# B&R Automation Studio project Panasonic_LinkaPowerCP2_A2021055 (part 15)

#### Main.st - Init, cyclic, exit code
```iecst
PROGRAM _INIT
	(* Insert code here *)

END_PROGRAM

PROGRAM _CYCLIC

	//*************************************Prepnutie obrazovky pri stlačení tlačítka CS*********************************//
	IF EDGEPOS(P1_Pracovisko.STAV.Manual AND NOT Safety.STAV.Linka_ZonaCS_AKTIVNA) THEN
		P1_Vizu.GoPage:= 'PageAutomatP1';
	END_IF

	//************************************Filter alarmov**************************************************************//
	FilterVizu_P1:= '[{"logicalOperator":"and","value":100,"conditionType":">=","columnType":"cod","useAlarmState":false,"alarmState":0},{"value":199,"conditionType":"<=","columnType":"cod","useAlarmState":false,"alarmState":0}]';

	//Zmeny farieb tlačítok ovládania zámkov//
	//Predné dvere //
	IF P1_Pracovisko.OUT.PredneDvere_ZAMKNI AND P1_Pracovisko.IN.PredneDvere_PritomnostAdaptera THEN
		P1_Vizu.TL_PrednyZamok_Farba:= "Button_Green";
	ELSIF P1_Pracovisko.IN.PredneDvere_PritomnostAdaptera THEN
		IF Blikac1s THEN
			P1_Vizu.TL_PrednyZamok_Farba:= "Button_Blue";
		ELSE
			P1_Vizu.TL_PrednyZamok_Farba:= "Operate";
		END_IF
	ELSE
		P1_Vizu.TL_PrednyZamok_Farba:= "Button_Red";
	END_IF

	//Zadné dvere//
	IF P1_Pracovisko.OUT.ZadneDvere_ZAMKNI AND P1_Pracovisko.IN.ZadneDvere_PritomnostAdaptera THEN
		P1_Vizu.TL_ZadnyZamok_Farba:= "Button_Green";
	ELSIF P1_Pracovisko.IN.ZadneDvere_PritomnostAdaptera THEN
		IF Blikac1s THEN
			P1_Vizu.TL_ZadnyZamok_Farba:= "Button_Blue";
		ELSE
			P1_Vizu.TL_ZadnyZamok_Farba:= "Operate";
		END_IF
	ELSE
		P1_Vizu.TL_ZadnyZamok_Farba:= "Button_Red";
	END_IF

	//***********************************Zobrazenie warningov pracoviska****************************************************//
	//0 - Pracovisko je vypnuté.
	//1 - Prebieha inicializácia pracoviska.
	//2 - Na pracovisku prebieha výroba.
	//3 - Prebieha ukončenie pracovného cyklu pracoviska.
	//4 - Prebieha režim vyprázdnenia linky.
	//5 - Robot nie je prepnuty do automatického režimu !!!
	//6 - Doplň zásobník skrutiek K30 !!!
	//7 - Doplň zásobník skrutiek M5 !!!
	//8 - Doplň zásobník skrutiek M4 !!!
	//10 - Testovací kus

	IF NOT P1_Robot.COM_IN.Stav_RezimAUTOMAT THEN
		P1_Vizu.Warnings_Index:= 5;
	ELSIF P1_Pracovisko.STAV.Automat AND NOT P1_Pracovisko.STAV.PoINIT AND NOT P1_Pracovisko.STAV.UkoncenieCyklu_BUSY THEN
		P1_Vizu.Warnings_Index:= 1;
	ELSIF P1_Srobovanie.SkrutSet_K30.IN.VibracnyHrniec.PritomnostSkrutiekVHrnci THEN
		P1_Vizu.Warnings_Index:= 6;
	ELSIF P1_Srobovanie.SkrutSet_M5.IN.ZasobnikSkrutiekPrazdny THEN
		P1_Vizu.Warnings_Index:= 7;
	ELSIF P1_Srobovanie.SkrutSet_M4.IN.ZasobnikSkrutiekPrazdny THEN
		P1_Vizu.Warnings_Index:= 8;
	ELSIF Linka.PAR.TestovaciKus THEN
		P1_Vizu.Warnings_Index:= 10;
	ELSIF Linka.PAR.VyprazdnenieLinky THEN
		P1_Vizu.Warnings_Index:= 4;
	ELSIF P1_Pracovisko.STAV.PoINIT AND NOT P1_Pracovisko.STAV.UkoncenieCyklu_BUSY THEN
		P1_Vizu.Warnings_Index:= 2;
	ELSIF P1_Pracovisko.STAV.UkoncenieCyklu_BUSY THEN
		P1_Vizu.Warnings_Index:= 3;
	ELSIF NOT P1_Pracovisko.STAV.Automat THEN
		P1_Vizu.Warnings_Index:= 0;
	END_IF

	//************************Prepínanie farby textového pola warning zariadenia***********************************//
	IF P1_Vizu.Warnings_Index = 0 THEN
		P1_Vizu.Warnings_Farba:= "TextOutput_Grey";
	ELSIF P1_Vizu.Warnings_Index = 1 THEN
		P1_Vizu.Warnings_Farba:= "TextOutput_Blue";
	ELSIF P1_Vizu.Warnings_Index = 2 THEN
		P1_Vizu.Warnings_Farba:= "TextOutput_Green";
	ELSIF P1_Vizu.Warnings_Index = 3 THEN
		P1_Vizu.Warnings_Farba:= "TextOutput_Blue";
	ELSIF P1_Vizu.Warnings_Index = 4 THEN
		P1_Vizu.Warnings_Farba:= "TextOutput_Green";
	ELSIF P1_Vizu.Warnings_Index = 10 THEN
		P1_Vizu.Warnings_Farba:= "TextOutput_Green";
	ELSE
		IF Blikac1s THEN
			P1_Vizu.Warnings_Farba:= "TextOutput_Orange";
		ELSE
			P1_Vizu.Warnings_Farba:= "TextOutput_Grey";
		END_IF
	END_IF

	//***********************Prepnutie bootovacej obrazovky********************************//
	IF P1_Vizu.ActualPage <> 'PageBootP1' AND NOT Safety.STAV.Linka_SafetyPLC_Nabehlo THEN
		P1_Vizu.GoPage:= 'PageBootP1';
	ELSIF P1_Vizu.ActualPage = 'PageBootP1' AND Safety.STAV.Linka_SafetyPLC_Nabehlo THEN
		P1_Vizu.GoPage:= 'PageAutomatP1';
	END_IF

	IF P1_Vizu.GoPage = 'PageBootP1' AND P1_Vizu.ActualPage = 'PageBootP1' THEN
		P1_Vizu.GoPage:= '';
	ELSIF P1_Vizu.GoPage = 'PageAutomatP1' AND P1_Vizu.ActualPage = 'PageAutomatP1' THEN
		P1_Vizu.GoPage:= '';
	END_IF

	//********************************Blikanie tlačítka Alarmy*******************************************************//
	IF P1_Pracovisko.STAV.PORUCHA AND P1_Vizu.ActualPage <> 'PageAlarmP1' THEN
		IF Blikac500ms THEN
			P1_AlarmyVizu.FarbaTlacitka_Alarmy:= "Button_Red";
		ELSE
			P1_AlarmyVizu.FarbaTlacitka_Alarmy:= "default";
		END_IF
	ELSE
		P1_AlarmyVizu.FarbaTlacitka_Alarmy:= "default";
	END_IF

	//*************************************Zamknutie tlačítok***************************************************************//
	//Zamknutie tlačítok ovládania zámkov//
	IF P1_Pracovisko.STAV.Automat THEN
		P1_Vizu.TL_OvladaniaZamkov_ENABLE:= FALSE;
	ELSIF P1_Srobovanie.STAV.RR_Polohovanie_BUSY THEN
		P1_Vizu.TL_OvladaniaZamkov_ENABLE:= FALSE;
	ELSIF P1_Srobovanie.STAV.CistenieSkrutkovackyK30_BUSY THEN
		P1_Vizu.TL_OvladaniaZamkov_ENABLE:= FALSE;
	ELSE
		P1_Vizu.TL_OvladaniaZamkov_ENABLE:= TRUE;
	END_IF

	//Tlačítko Štat Automat//
	IF P1_Pracovisko.STAV.UkoncenieCyklu_BUSY THEN
		P1_Vizu.TL_StartAutomat_ENABLE:= FALSE;
	ELSIF P1_Pracovisko.STAV.PORUCHA THEN
		P1_Vizu.TL_StartAutomat_ENABLE:= FALSE;
	ELSIF NOT P1_Robot.COM_IN.Stav_RezimAUTOMAT THEN
		P1_Vizu.TL_StartAutomat_ENABLE:= FALSE;
	ELSIF NOT Safety.STAV.P1_ZonaBunky_AKTIVNA THEN
		P1_Vizu.TL_StartAutomat_ENABLE:= FALSE;
	ELSIF NOT P1_Pracovisko.STAV.HardwareVytahu_OK THEN
		P1_Vizu.TL_StartAutomat_ENABLE:= FALSE;
	ELSIF NOT P1_Pracovisko.STAV.HardwareBunky_OK THEN
		P1_Vizu.TL_StartAutomat_ENABLE:= FALSE;
	ELSE
		P1_Vizu.TL_StartAutomat_ENABLE:= TRUE;
	END_IF

	//Tlačítko Ukončenie Cyklu//
	IF P1_Pracovisko.STAV.PoINIT THEN
		P1_Vizu.TL_KoniecCyklu_ENABLE:= TRUE;
	ELSE
		P1_Vizu.TL_KoniecCyklu_ENABLE:= FALSE;
	END_IF

	//Tlačítko STOP//
	IF P1_Pracovisko.STAV.PoINIT AND NOT P1_Pracovisko.STAV.UkoncenieCyklu_BUSY THEN
		P1_Vizu.TL_STOP_ENABLE:= FALSE;
	ELSE
		P1_Vizu.TL_STOP_ENABLE:= TRUE;
	END_IF

	//Tlačítko Režim Automat//

	P1_Vizu.TL_RezimAutomat_ENABLE:= TRUE;

	//Tlačítko Režim Manual//
	IF P1_Pracovisko.STAV.Automat THEN
		P1_Vizu.TL_RezimManual_ENABLE:= FALSE;
	ELSIF NOT P1_Pracovisko.STAV.HardwareVytahu_OK THEN
		P1_Vizu.TL_RezimManual_ENABLE:= FALSE;
	ELSIF NOT P1_Pracovisko.STAV.HardwareBunky_OK THEN
		P1_Vizu.TL_RezimManual_ENABLE:= FALSE;
	ELSE
		P1_Vizu.TL_RezimManual_ENABLE:= TRUE;
	END_IF

	//Tlačítko zmena modelu//
	IF Linka.STAV.OFF THEN
		P1_Vizu.TL_VolbaModelu_ENABLE:= TRUE;
	ELSE
		P1_Vizu.TL_VolbaModelu_ENABLE:= FALSE;
	END_IF

	//Tlačítko paletka prechádza//
	IF NOT Linka.STAV.PoINIT THEN
		P1_Vizu.TL_PaletkaPrechadza_ENABLE:= FALSE;
	ELSIF NOT P1_Vytah.RFID_hlava.PritomnostPaletky THEN
		P1_Vizu.TL_PaletkaPrechadza_ENABLE:= FALSE;
	ELSIF Linka.PAR.TestovaciKus THEN
		P1_Vizu.TL_PaletkaPrechadza_ENABLE:= FALSE;
	ELSIF Linka.PAR.RevorkovyKus THEN
		P1_Vizu.TL_PaletkaPrechadza_ENABLE:= FALSE;
	ELSIF Linka.PAR.PaletkaPrechadza THEN
		P1_Vizu.TL_PaletkaPrechadza_ENABLE:= FALSE;
	ELSE
		P1_Vizu.TL_PaletkaPrechadza_ENABLE:= TRUE;
	END_IF

	//Tlačítko vyprázdnenie linky//
	IF Linka.PAR.VyprazdnenieLinky THEN
		P1_Vizu.TL_VyprazdnenieLinky_ENABLE:= FALSE;
	ELSIF NOT P4_Pracovisko.STAV.Automat THEN
		P1_Vizu.TL_VyprazdnenieLinky_ENABLE:= FALSE;
	ELSIF Linka.PAR.TestovaciKus THEN
		P1_Vizu.TL_VyprazdnenieLinky_ENABLE:= FALSE;
	ELSE
		P1_Vizu.TL_VyprazdnenieLinky_ENABLE:= TRUE;
	END_IF

	//Tlačítko testovací kus//
	IF NOT Linka.STAV.PoINIT THEN
		P1_Vizu.TL_TestovaciKus_ENABLE:= FALSE;
	ELSIF Linka.PAR.RevorkovyKus THEN
		P1_Vizu.TL_TestovaciKus_ENABLE:= FALSE;
	ELSIF NOT P1_Vytah.RFID_hlava.PritomnostPaletky THEN
		P1_Vizu.TL_TestovaciKus_ENABLE:= FALSE;
	ELSIF Linka.PAR.PaletkaPrechadza THEN
		P1_Vizu.TL_TestovaciKus_ENABLE:= FALSE;
	ELSE
		P1_Vizu.TL_TestovaciKus_ENABLE:= TRUE;
	END_IF

	//Tlačítko revork//
	IF NOT Linka.STAV.PoINIT THEN
		P1_Vizu.TL_Revork_ENABLE:= FALSE;
	ELSIF NOT P1_Vytah.RFID_hlava.PritomnostPaletky THEN
		P1_Vizu.TL_Revork_ENABLE:= FALSE;
	ELSIF Linka.PAR.TestovaciKus THEN
		P1_Vizu.TL_Revork_ENABLE:= FALSE;
	ELSIF Linka.PAR.PaletkaPrechadza THEN
		P1_Vizu.TL_Revork_ENABLE:= FALSE;
	ELSE
		P1_Vizu.TL_Revork_ENABLE:= TRUE;
	END_IF

	//Tlačítko výtah čítanie paletky//
	IF P1_Vytah.RFID_hlava.PritomnostPaletky THEN
		P1_Vizu.Vytah_CitaniePaletky_ENABLE:= TRUE;
	ELSE
		P1_Vizu.Vytah_CitaniePaletky_ENABLE:= FALSE;
	END_IF

	//Tlačítko výťah zápis paletky//
	IF P1_Vytah.RFID_hlava.PritomnostPaletky THEN
		P1_Vizu.Vytah_ZapisPaletky_ENABLE:= TRUE;
	ELSE
		P1_Vizu.Vytah_ZapisPaletky_ENABLE:= FALSE;
	END_IF

	//RR - Tlačítko čistenia skrutkovačky K30//
	IF P1_Srobovanie.STAV.RR_Polohovanie_BUSY THEN
		P1_Vizu.TL_VycistiSkrutkovackuK30_ENABLE:= FALSE;
	ELSIF NOT Safety.STAV.P1_ZonaBunky_AKTIVNA THEN
		P1_Vizu.TL_VycistiSkrutkovackuK30_ENABLE:= FALSE;
	ELSIF NOT Safety.STAV.Linka_ZonaCS_AKTIVNA THEN
		P1_Vizu.TL_VycistiSkrutkovackuK30_ENABLE:= FALSE;
	ELSIF P1_Srobovanie.STAV.CistenieSkrutkovackyK30_BUSY THEN
		P1_Vizu.TL_VycistiSkrutkovackuK30_ENABLE:= FALSE;
	ELSIF NOT P1_Pracovisko.STAV.SkrutkovackyZasunute THEN
		P1_Vizu.TL_VycistiSkrutkovackuK30_ENABLE:= FALSE;
	ELSIF P1_Srobovanie.CMD.RR_SkrutSetK30_VysunBrzdu THEN
		P1_Vizu.TL_VycistiSkrutkovackuK30_ENABLE:= FALSE;
	ELSIF P1_Srobovanie.CMD.RR_SkrutSetK30_Zasobnik_RUN THEN
		P1_Vizu.TL_VycistiSkrutkovackuK30_ENABLE:= FALSE;
	ELSE
		P1_Vizu.TL_VycistiSkrutkovackuK30_ENABLE:= TRUE;
	END_IF

	//RR - Tlačítko polohovania aplikátora//
	IF P1_Srobovanie.STAV.RR_Polohovanie_BUSY THEN
		P1_Vizu.TL_PolohujManipulator_ENABLE:= FALSE;
	ELSIF NOT Safety.STAV.P1_ZonaBunky_AKTIVNA THEN
		P1_Vizu.TL_PolohujManipulator_ENABLE:= FALSE;
	ELSIF NOT Safety.STAV.Linka_ZonaCS_AKTIVNA THEN
		P1_Vizu.TL_PolohujManipulator_ENABLE:= FALSE;
	ELSIF P1_Srobovanie.STAV.CistenieSkrutkovackyK30_BUSY THEN
		P1_Vizu.TL_PolohujManipulator_ENABLE:= FALSE;
	ELSIF NOT P1_Pracovisko.STAV.SkrutkovackyZasunute THEN
		P1_Vizu.TL_PolohujManipulator_ENABLE:= FALSE;
	ELSE
		P1_Vizu.TL_PolohujManipulator_ENABLE:= TRUE;
	END_IF

	//RR - Tlačítko vysunutia skrutkovačky K30//
	IF P1_Srobovanie.STAV.RR_Polohovanie_BUSY THEN
		P1_Vizu.Tl_VysunutieSkrutkovK30_ENABLE:= FALSE;
	ELSIF P1_Srobovanie.STAV.CistenieSkrutkovackyK30_BUSY THEN
		P1_Vizu.Tl_VysunutieSkrutkovK30_ENABLE:= FALSE;
	ELSIF NOT Safety.STAV.P1_ZonaBunky_AKTIVNA THEN
		P1_Vizu.Tl_VysunutieSkrutkovK30_ENABLE:= FALSE;
	ELSIF NOT Safety.STAV.Linka_ZonaCS_AKTIVNA THEN
		P1_Vizu.Tl_VysunutieSkrutkovK30_ENABLE:= FALSE;
	ELSE
		P1_Vizu.Tl_VysunutieSkrutkovK30_ENABLE:= TRUE;
	END_IF

	//RR - Tlačítko vysunutia skrutkovačiek M4 a M5//
	IF P1_Srobovanie.STAV.RR_Polohovanie_BUSY THEN
		P1_Vizu.TL_OvladaniaVysunSkrutkovM4_M5:= FALSE;
	ELSIF P1_Srobovanie.STAV.CistenieSkrutkovackyK30_BUSY THEN
		P1_Vizu.TL_OvladaniaVysunSkrutkovM4_M5:= FALSE;
	ELSIF NOT Safety.STAV.P1_ZonaBunky_AKTIVNA THEN
		P1_Vizu.TL_OvladaniaVysunSkrutkovM4_M5:= FALSE;
	ELSIF NOT Safety.STAV.Linka_ZonaCS_AKTIVNA THEN
		P1_Vizu.TL_OvladaniaVysunSkrutkovM4_M5:= FALSE;
	ELSE
		P1_Vizu.TL_OvladaniaVysunSkrutkovM4_M5:= TRUE;
	END_IF

	//RR - Ovládanie skrutkovacieho setu//
	IF P1_Srobovanie.STAV.CistenieSkrutkovackyK30_BUSY THEN
		P1_Vizu.TL_OvladSkrutkovSetuK30_ENABLE:= FALSE;
	ELSE
		P1_Vizu.TL_OvladSkrutkovSetuK30_ENABLE:= TRUE;
	END_IF

	//RR - Ovládanie manipulatora XY//
	IF NOT Safety.STAV.P1_ZonaBunky_AKTIVNA THEN
		P1_Vizu.TL_OvladManipulatoraXY_ENABLE:= FALSE;
	ELSE
		P1_Vizu.TL_OvladManipulatoraXY_ENABLE:= TRUE;
	END_IF

	//**************************Zamknutie editácie parametrov*********************************//
	IF P1_UrovenPrihlasenehoUzivatela >= 20 THEN
		P1_Vizu.EditaciaParametrov_ENABLE:= TRUE;
	ELSE
		P1_Vizu.EditaciaParametrov_ENABLE:= FALSE;
	END_IF

	//***********************************Prepínanie stavov pracovísk*******************************************************************//
	//Výťah//
	IF NOT P1_Pracovisko.STAV.HardwareVytahu_OK THEN
		P1_Vizu.IndexStavu_Vytah:= 3;
	ELSIF P1_Pracovisko.STAV.Porucha_ST1 THEN
		P1_Vizu.IndexStavu_Vytah:= 3;
	ELSIF P1_Vytah.Automat AND NOT P1_Vytah.STAV.PoINIT THEN
		P1_Vizu.IndexStavu_Vytah:= 1;
	ELSIF P1_Vytah.Automat AND P1_Vytah.STAV.PoINIT THEN
		P1_Vizu.IndexStavu_Vytah:= 2;
	ELSE
		P1_Vizu.IndexStavu_Vytah:= 0;
	END_IF

	//Dopravníky//
	IF P1_Dopravniky.Automat AND NOT P1_Dopravniky.STAV.PoINIT THEN
		P1_Vizu.IndexStavu_Dopravnik:= 1;
	ELSIF P1_Dopravniky.Automat AND P1_Dopravniky.STAV.PoINIT THEN
		P1_Vizu.IndexStavu_Dopravnik:= 2;
	ELSE
		P1_Vizu.IndexStavu_Dopravnik:= 0;
	END_IF

	//Spodný stoper//
	IF P1_SpodnyStoper.Automat AND NOT P1_SpodnyStoper.STAV.PoINIT THEN
		P1_Vizu.IndexStavu_SpodnyStoper:= 1;
	ELSIF P1_SpodnyStoper.Automat AND P1_SpodnyStoper.STAV.PoINIT THEN
		P1_Vizu.IndexStavu_SpodnyStoper:= 2;
	ELSE
		P1_Vizu.IndexStavu_SpodnyStoper:= 0;
	END_IF

	//Stoper šrobovania//
	IF NOT P1_Pracovisko.STAV.HardwareBunky_OK THEN
		P1_Vizu.IndexStavu_StoperSrobovania:= 3;
	ELSIF P1_Pracovisko.STAV.Porucha_ST2 THEN
		P1_Vizu.IndexStavu_StoperSrobovania:= 3;
	ELSIF P1_StoperSrobovania.Automat AND NOT P1_StoperSrobovania.STAV.PoINIT THEN
		P1_Vizu.IndexStavu_StoperSrobovania:= 1;
	ELSIF P1_StoperSrobovania.Automat AND P1_StoperSrobovania.STAV.PoINIT THEN
		P1_Vizu.IndexStavu_StoperSrobovania:= 2;
	ELSE
		P1_Vizu.IndexStavu_StoperSrobovania:= 0;
	END_IF

	//Šrobovanie//
	IF NOT P1_Pracovisko.STAV.HardwareBunky_OK THEN
		P1_Vizu.IndexStavu_Srobovanie:= 3;
	ELSIF P1_Pracovisko.STAV.Porucha_ST2 THEN
		P1_Vizu.IndexStavu_Srobovanie:= 3;
	ELSIF P1_Srobovanie.Automat AND NOT P1_Srobovanie.STAV.PoINIT THEN
		P1_Vizu.IndexStavu_Srobovanie:= 1;
	ELSIF P1_Srobovanie.Automat AND P1_Srobovanie.STAV.PoINIT THEN
		P1_Vizu.IndexStavu_Srobovanie:= 2;
	ELSE
		P1_Vizu.IndexStavu_Srobovanie:= 0;
	END_IF

	//Akumulačný stoper//
	IF P1_Pracovisko.STAV.Porucha_ST3 THEN
		P1_Vizu.IndexStavu_AkumulacnyStoper:= 3;
	ELSIF P1_AkumulacnyStoper.Automat AND NOT P1_AkumulacnyStoper.STAV.PoINIT THEN
		P1_Vizu.IndexStavu_AkumulacnyStoper:= 1;
	ELSIF P1_AkumulacnyStoper.Automat AND P1_AkumulacnyStoper.STAV.PoINIT THEN
		P1_Vizu.IndexStavu_AkumulacnyStoper:= 2;
	ELSE
		P1_Vizu.IndexStavu_AkumulacnyStoper:= 0;
	END_IF

	//Robot//
	IF P1_Robot.Automat AND NOT P1_Robot.STAV.PoINIT THEN
		P1_Vizu.IndexStavu_Robot:= 1;
	ELSIF P1_Robot.Automat AND P1_Robot.STAV.PoINIT THEN
		P1_Vizu.IndexStavu_Robot:= 2;
	ELSE
		P1_Vizu.IndexStavu_Robot:= 0;
	END_IF

END_PROGRAM

PROGRAM _EXIT
	(* Insert code here *)

END_PROGRAM
```

### Program Logical/Program/Pracovisko_1/P1_OvladSafety (IEC)

#### Main.st - Init, cyclic, exit code
```iecst
PROGRAM _INIT
	(* Insert code here *)

END_PROGRAM

PROGRAM _CYCLIC

	//******************************************Ovládanie zámkov dverí bunky****************************************//
	//Predné dvere //
	IF P1_Vizu.TL_ZamkniPrednyZamok THEN
		IF NOT P1_Pracovisko.OUT.PredneDvere_ZAMKNI AND P1_Pracovisko.IN.PredneDvere_PritomnostAdaptera THEN
			P1_Pracovisko.OUT.PredneDvere_ZAMKNI:= TRUE;
		ELSIF P1_Pracovisko.OUT.PredneDvere_ZAMKNI THEN
			P1_Pracovisko.OUT.PredneDvere_ZAMKNI:= FALSE;
		END_IF
		P1_Vizu.TL_ZamkniPrednyZamok:= FALSE;
	END_IF

	//Zadné dvere//
	IF P1_Vizu.TL_ZamkniZadnyZamok THEN
		IF NOT P1_Pracovisko.OUT.ZadneDvere_ZAMKNI AND P1_Pracovisko.IN.ZadneDvere_PritomnostAdaptera THEN
			P1_Pracovisko.OUT.ZadneDvere_ZAMKNI:= TRUE;
		ELSIF P1_Pracovisko.OUT.ZadneDvere_ZAMKNI THEN
			P1_Pracovisko.OUT.ZadneDvere_ZAMKNI:= FALSE;
		END_IF
		P1_Vizu.TL_ZamkniZadnyZamok:= FALSE;
	END_IF

	//******************************************Reset zóny výtahu*********************************************//
	IF Safety.STAV.Linka_ZonaCS_AKTIVNA AND
		(Safety.STAV.P1_Vytah_Bariera_AKTIVNA OR Safety.STAV.P1_Vytah_Muting_AKTIVNY) AND
		NOT Safety.STAV.P1_ZonaVytahu_AKTIVNA THEN
		Safety.OUT.P1_ResetZonyVytahu:= TRUE;
	ELSE
		Safety.OUT.P1_ResetZonyVytahu:= FALSE;
	END_IF

	//*****************************************Reset zóny bunky************************************************//
	IF Safety.STAV.Linka_ZonaCS_AKTIVNA AND
		(Safety.STAV.P1_Bunka_Zamky_AKTIVNE OR Safety.STAV.P1_VyblokovanieZamkov_AKTIVNE) AND
		NOT Safety.STAV.P1_ZonaBunky_AKTIVNA AND
		(Safety.STAV.P1_VstupBunky_VstupBar_AKTIVNA OR Safety.STAV.P1_VstupBunky_VystupBar_AKTIVNA) AND
		(Safety.STAV.P1_VystupBunky_VstupBar_AKTIVNA OR Safety.STAV.P1_VystupBunky_VystupBar_AKTIVNA) THEN
		Safety.OUT.P1_ResetZonyBunky:= TRUE;
	ELSE
		Safety.OUT.P1_ResetZonyBunky:= FALSE;
	END_IF

END_PROGRAM

PROGRAM _EXIT
	(* Insert code here *)

END_PROGRAM
```

### Program Logical/Program/Pracovisko_1/P1_Mapping_IO (IEC)

#### Main.st - Init, cyclic, exit code
```iecst
PROGRAM _INIT
	(* Insert code here *)

END_PROGRAM

PROGRAM _CYCLIC

	//**********************************************************IO modul Wedmuller**********************************************************************//
	//************Karta AB 1.2 8DI**************//
	P1_Srobovanie.IN.NapajanieSkrutkovackyK30_OK :=  P1_Pracovisko.COM_Weidmuller.AB1_2_8DI.0;
	P1_Srobovanie.IN.NapajanieSkrutkovackyM5_OK := P1_Pracovisko.COM_Weidmuller.AB1_2_8DI.1;
	P1_Srobovanie.IN.NapajanieSkrutkovackyM4_OK := P1_Pracovisko.COM_Weidmuller.AB1_2_8DI.2;
	P1_Srobovanie.IN.NapajanieZasobnikaM4_OK := P1_Pracovisko.COM_Weidmuller.AB1_2_8DI.3;
	P1_Srobovanie.IN.NapajanieVibrolistyM4_OK := P1_Pracovisko.COM_Weidmuller.AB1_2_8DI.4;
	P1_Srobovanie.IN.NapajanieZasobnikaM5_OK := P1_Pracovisko.COM_Weidmuller.AB1_2_8DI.5;
	P1_Srobovanie.IN.NapajanieVibrolistyM5_OK := P1_Pracovisko.COM_Weidmuller.AB1_2_8DI.6;
	P1_Vytah.IN.StavRiadeniaDopravVytahu_READY := P1_Pracovisko.COM_Weidmuller.AB1_2_8DI.7;

	//***********Karta AB 1.3 8DI***************//
	P1_Dopravniky.IN.StavRiadeniaDopravBunky_READY := P1_Pracovisko.COM_Weidmuller.AB1_3_8DI.0;
	P1_Dopravniky.IN.StavRiadeniaVratnehoDoprav_READY := P1_Pracovisko.COM_Weidmuller.AB1_3_8DI.1;
	P1_Vytah.IN.TeplotaMotoraDopravVytahu_OK := P1_Pracovisko.COM_Weidmuller.AB1_3_8DI.2;
	P1_Dopravniky.IN.TeplotaMotoraDopravBunky_OK := P1_Pracovisko.COM_Weidmuller.AB1_3_8DI.3;
	P1_Dopravniky.IN.TeplotaMotoraVratnehoDoprav_OK := P1_Pracovisko.COM_Weidmuller.AB1_3_8DI.4;
	P1_Pracovisko.COM_Weidmuller.AB1_3_8DI.5;
	P1_Pracovisko.COM_Weidmuller.AB1_3_8DI.6;
	P1_Srobovanie.IN.NapajanieZasobnikaK30_OK := P1_Pracovisko.COM_Weidmuller.AB1_3_8DI.7;

	//************Karta AB 1.4 8DI**************//
	P1_Pracovisko.COM_Weidmuller.AB1_4_8DI.0;
	P1_Pracovisko.COM_Weidmuller.AB1_4_8DI.1;
	P1_Pracovisko.COM_Weidmuller.AB1_4_8DI.2;
	P1_Pracovisko.COM_Weidmuller.AB1_4_8DI.3;
	P1_Pracovisko.COM_Weidmuller.AB1_4_8DI.4;
	P1_Pracovisko.COM_Weidmuller.AB1_4_8DI.5;
	P1_Pracovisko.COM_Weidmuller.AB1_4_8DI.6;
	P1_Pracovisko.COM_Weidmuller.AB1_4_8DI.7;

	//************Karta AB 1.5 8DI***************//
	Safety.IN.Linka_SV_ZonaCS := P1_Pracovisko.COM_Weidmuller.AB1_5_8DI.0;
	Safety.IN.P1_SV_ZonaBunky := P1_Pracovisko.COM_Weidmuller.AB1_5_8DI.1;
	Safety.IN.P1_SV_ZonaVytahu := P1_Pracovisko.COM_Weidmuller.AB1_5_8DI.2;
	P1_Pracovisko.COM_Weidmuller.AB1_5_8DI.3;
	P1_Pracovisko.COM_Weidmuller.AB1_5_8DI.4;
	P1_Pracovisko.COM_Weidmuller.AB1_5_8DI.5;
	P1_Pracovisko.COM_Weidmuller.AB1_5_8DI.6;
	P1_Pracovisko.COM_Weidmuller.AB1_5_8DI.7;

	//************Karta AB 1.6 8DO***************//
	P1_Pracovisko.COM_Weidmuller.AB1_6_8DO.0 := P1_Pracovisko.OUT.Majak_ZeleneSvetlo_ON;
	P1_Pracovisko.COM_Weidmuller.AB1_6_8DO.1 := P1_Pracovisko.OUT.Majak_OranzoveSvetlo_ON;
	P1_Pracovisko.COM_Weidmuller.AB1_6_8DO.2 := P1_Pracovisko.OUT.Majak_CerveneSvetlo_ON;
	P1_Pracovisko.COM_Weidmuller.AB1_6_8DO.3 := P1_Pracovisko.OUT.Majak_Hukacka_ON;
	P1_Pracovisko.COM_Weidmuller.AB1_6_8DO.4 := P1_Srobovanie.SkrutSet_M4.OUT.VibropohonZasobnika_RUN;
	P1_Pracovisko.COM_Weidmuller.AB1_6_8DO.5 := P1_Srobovanie.SkrutSet_M4.OUT.VibropohonListy_RUN;
	P1_Pracovisko.COM_Weidmuller.AB1_6_8DO.6 := P1_Srobovanie.SkrutSet_M5.OUT.VibropohonZasobnika_RUN;
	P1_Pracovisko.COM_Weidmuller.AB1_6_8DO.7 := P1_Srobovanie.SkrutSet_M5.OUT.VibropohonListy_RUN;

	//************Karta AB 1.7 8DO***************//
	P1_Pracovisko.COM_Weidmuller.AB1_7_8DO.0 := P1_Pracovisko.OUT.OsvetlenieBunky_ON;
	P1_Pracovisko.COM_Weidmuller.AB1_7_8DO.1 := P1_Vytah.OUT.DopravnikChod_VPRED;
	P1_Pracovisko.COM_Weidmuller.AB1_7_8DO.2 := P1_Vytah.OUT.DopravnikChod_VZAD;
	P1_Pracovisko.COM_Weidmuller.AB1_7_8DO.3 := P1_Dopravniky.OUT.DopravnikBunky_ON;
	P1_Pracovisko.COM_Weidmuller.AB1_7_8DO.4 := P1_Dopravniky.OUT.VratnyDopravnik_ON;
	P1_Pracovisko.COM_Weidmuller.AB1_7_8DO.5 := P1_Robot.OUT.Griper_OTVOR;
	P1_Pracovisko.COM_Weidmuller.AB1_7_8DO.6 := P1_Robot.OUT.Griper_ZATVOR;
	P1_Pracovisko.COM_Weidmuller.AB1_7_8DO.7;

	//***********Karta AB 1.9 8DO*****************//
	P1_Pracovisko.COM_Weidmuller.AB1_9_8DO.0;
	P1_Pracovisko.COM_Weidmuller.AB1_9_8DO.1;
	P1_Pracovisko.COM_Weidmuller.AB1_9_8DO.2;
	P1_Pracovisko.COM_Weidmuller.AB1_9_8DO.3;
	P1_Pracovisko.COM_Weidmuller.AB1_9_8DO.4:= P1_Vytah.OUT.OsvetlenieVytahu_ON;
	P1_Pracovisko.COM_Weidmuller.AB1_9_8DO.5:= P1_Pracovisko.OUT.Osvetlenie_CAM4_ON;
	P1_Pracovisko.COM_Weidmuller.AB1_9_8DO.6:= P1_Pracovisko.OUT.Osvetlenie_CAM6_ON;
	P1_Pracovisko.COM_Weidmuller.AB1_9_8DO.7 := P1_Srobovanie.SkrutSet_K30.OUT.VibracnyHrniec.ZapniVibromotor; (*SkrutkSet_K30.OUT.VibropohonZasobnika_RUN;*)

	//**********Karta AB 1.10 8DO***************//
	P1_Pracovisko.COM_Weidmuller.AB1_10_8DO.0:= Safety.OUT.Linka_ResetCS;
	P1_Pracovisko.COM_Weidmuller.AB1_10_8DO.1:= Safety.OUT.P1_ResetZonyBunky;
	P1_Pracovisko.COM_Weidmuller.AB1_10_8DO.2:= Safety.OUT.P1_ResetZonyVytahu;
	P1_Pracovisko.COM_Weidmuller.AB1_10_8DO.3; //Safety resety
	P1_Pracovisko.COM_Weidmuller.AB1_10_8DO.4:= P1_Pracovisko.OUT.Srobovanie_OsvetleniePaletky_ON;
	P1_Pracovisko.COM_Weidmuller.AB1_10_8DO.5:= P1_Pracovisko.OUT.Srobovanie_BodoveOsvetlenie_ON;
	P1_Pracovisko.COM_Weidmuller.AB1_10_8DO.6;
	P1_Pracovisko.COM_Weidmuller.AB1_10_8DO.7;

	//**************************************************************IO modul Festo**********************************************************************************//

	//**********Modul DM 1.1 4DI4DO**************//
	//Inputs//
	P1_Pracovisko.IN.PredneDvere_PritomnostAdaptera := P1_Pracovisko.COM_Festo.DM1_1_4DI[0];
	P1_Pracovisko.IN.ZadneDvere_PritomnostAdaptera := P1_Pracovisko.COM_Festo.DM1_1_4DI[1];
	P1_Pracovisko.COM_Festo.DM1_1_4DI[2];
	P1_Pracovisko.COM_Festo.DM1_1_4DI[3];

	//Outputs//
	P1_Pracovisko.COM_Festo.DM1_1_4DO[0]:= P1_Pracovisko.OUT.PredneDvere_ZAMKNI ;
	P1_Pracovisko.COM_Festo.DM1_1_4DO[1]:= P1_Pracovisko.OUT.ZadneDvere_ZAMKNI;
	P1_Pracovisko.COM_Festo.DM1_1_4DO[2];
	P1_Pracovisko.COM_Festo.DM1_1_4DO[3];

	//***********Modul DI 1.1 8DI****************//
	P1_StoperSrobovania.IN.Centrovanie_VYSUNUTE := P1_Pracovisko.COM_Festo.DI1_1_8DI[0];
	P1_StoperSrobovania.IN.Centrovanie_ZASUNUTE := P1_Pracovisko.COM_Festo.DI1_1_8DI[1];
	P1_AkumulacnyStoper.IN.PritomnostPaletky := P1_Pracovisko.COM_Festo.DI1_1_8DI[2];
	P1_SpodnyStoper.IN.PritomnostPaletky := P1_Pracovisko.COM_Festo.DI1_1_8DI[3];
	P1_SpodnyStoper.IN.ZaplnenieDopravnika := P1_Pracovisko.COM_Festo.DI1_1_8DI[4];
	P1_Robot.IN.Vakum_OK := P1_Pracovisko.COM_Festo.DI1_1_8DI[5];
	P1_Robot.IN.DokStanica_PritomnGripra5H := P1_Pracovisko.COM_Festo.DI1_1_8DI[6];
	P1_Robot.IN.DokStanica_PritomnGripra45F := P1_Pracovisko.COM_Festo.DI1_1_8DI[7];

	//************Modul DI 1.2 8DI***************//
	P1_Srobovanie.SkrutSet_M4.IN.ZasobnikSkrutiekPrazdny := P1_Pracovisko.COM_Festo.DI1_2_8DI[0];
	P1_Srobovanie.SkrutSet_M4.IN.ZaplnenieListyZasobnika := P1_Pracovisko.COM_Festo.DI1_2_8DI[1];
	P1_Srobovanie.SkrutSet_M4.IN.ZaplnenieVibrolisty_MAX := P1_Pracovisko.COM_Festo.DI1_2_8DI[2];
	P1_Srobovanie.SkrutSet_M4.IN.ZaplnenieVibrolisty_MIN := P1_Pracovisko.COM_Festo.DI1_2_8DI[3];
	P1_Srobovanie.SkrutSet_M4.IN.Podavac_SkrutkaNaVstupe := P1_Pracovisko.COM_Festo.DI1_2_8DI[4];
	P1_Srobovanie.SkrutSet_M4.IN.Podavac_SkrutkaNaVystupe := P1_Pracovisko.COM_Festo.DI1_2_8DI[5];
	P1_Srobovanie.SkrutSet_M4.IN.PodavacOtoceny_VSTUP := P1_Pracovisko.COM_Festo.DI1_2_8DI[6];
	P1_Srobovanie.SkrutSet_M4.IN.PodavacOtoceny_VYSTUP := P1_Pracovisko.COM_Festo.DI1_2_8DI[7];

	//************Modul DI 1.3 8DI**************//
	P1_Srobovanie.SkrutSet_K30.IN.VibracnyHrniec.PritomnostSkrutiekVHrnci := P1_Pracovisko.COM_Festo.DI1_3_8DI[0];   (*SkrutkSet_K30.IN.ZasobnikSkrutiekPrazdny*)
	P1_Srobovanie.SkrutSet_K30.IN.VibracnyHrniec.VibracnaListaZaplnena := P1_Pracovisko.COM_Festo.DI1_3_8DI[1]; (*SkrutkSet_K30.IN.ZaplnenieListyZasobnika*)
	P1_Srobovanie.SkrutSet_K30.IN.Brzda.PreletSkrutky := P1_Pracovisko.COM_Festo.DI1_3_8DI[2]; (*SkrutkSet_K30.IN.PreletSnimacPredSkrutkovackou*)
	P1_Srobovanie.SkrutSet_K30.IN.Brzda.SkrutkaPritomnaVBrzde := P1_Pracovisko.COM_Festo.DI1_3_8DI[3]; (*SkrutkSet_K30.IN.PreletSnimacPredBrzdou*)
	P1_Srobovanie.SkrutSet_K30.IN.Brzda.ZakladnaPoloha := P1_Pracovisko.COM_Festo.DI1_3_8DI[4]; //Brzda je zasunutá, vstup skrutky do brzdy     (*SkrutkSet_K30.IN.BrzdaZASUNUTA*)
	P1_Srobovanie.SkrutSet_K30.IN.Brzda.PodajSkrutku  := P1_Pracovisko.COM_Festo.DI1_3_8DI[5]; //Brzda je vysunuta, výstup skrutky s brzdy      (*SkrutkSet_K30.IN.BrzdaVYSUNUTA*)
	P1_Srobovanie.SkrutSet_K30.IN.VibracnyHrniec.PreletovySnimac  := P1_Pracovisko.COM_Festo.DI1_3_8DI[6];  (*SkrutkSet_K30.IN.PreletSnimacZaOddelovacom*)
	P1_Srobovanie.IN.Skrutkovacka_K30_ZASUNUTA := P1_Pracovisko.COM_Festo.DI1_3_8DI[7];   (*SkrutkSet_K30.IN.SkrutkovackaZASUNUTA*)

	//*************Modul DI 1.4 8DI**************//
	P1_Srobovanie.SkrutSet_M5.IN.ZasobnikSkrutiekPrazdny := P1_Pracovisko.COM_Festo.DI1_4_8DI[0];
	P1_Srobovanie.SkrutSet_M5.IN.ZaplnenieListyZasobnika := P1_Pracovisko.COM_Festo.DI1_4_8DI[1];
	P1_Srobovanie.SkrutSet_M5.IN.ZaplnenieVibrolisty_MAX := P1_Pracovisko.COM_Festo.DI1_4_8DI[2];
	P1_Srobovanie.SkrutSet_M5.IN.ZaplnenieVibrolisty_MIN := P1_Pracovisko.COM_Festo.DI1_4_8DI[3];
	P1_Srobovanie.SkrutSet_M5.IN.Podavac_SkrutkaNaVstupe := P1_Pracovisko.COM_Festo.DI1_4_8DI[4];
	P1_Srobovanie.SkrutSet_M5.IN.Podavac_SkrutkaNaVystupe := P1_Pracovisko.COM_Festo.DI1_4_8DI[5];
	P1_Srobovanie.SkrutSet_M5.IN.PodavacOtoceny_VSTUP := P1_Pracovisko.COM_Festo.DI1_4_8DI[6];
	P1_Srobovanie.SkrutSet_M5.IN.PodavacOtoceny_VYSTUP := P1_Pracovisko.COM_Festo.DI1_4_8DI[7];

	//**************Modul DI 1.5 8DI***************//
	P1_Vytah.IN.PrechodDopravnika := P1_Pracovisko.COM_Festo.DI1_5_8DI[0];
	P1_Pracovisko.IN.TlakVzduchu_OK := P1_Pracovisko.COM_Festo.DI1_5_8DI[1];
	Safety.IN.P1_SV_PrivodVzduchu_CH1 := P1_Pracovisko.COM_Festo.DI1_5_8DI[2];
	Safety.IN.P1_SV_PrivodVzduchu_CH2 := P1_Pracovisko.COM_Festo.DI1_5_8DI[3];
	P1_Srobovanie.IN.Skrutkovacka_M5_Vakum_OK := P1_Pracovisko.COM_Festo.DI1_5_8DI[4];
	P1_Srobovanie.IN.Skrutkovacka_M4_Vakum_OK := P1_Pracovisko.COM_Festo.DI1_5_8DI[5];
	P1_Pracovisko.COM_Festo.DI1_5_8DI[6];
	P1_Pracovisko.COM_Festo.DI1_5_8DI[7];

	//********Modul DS 1.1 IO link Port 0 - IO_Modul Balluff***************//
	//Inputs//
	P1_Robot.IN.Griper45F_Otvoreny:= P1_Pracovisko.COM_Festo.DS1_1_Port0_IN[0].0;
	P1_Robot.IN.Griper45F_Zatvoreny:= P1_Pracovisko.COM_Festo.DS1_1_Port0_IN[0].1;
	P1_Pracovisko.COM_Festo.DS1_1_Port0_IN[0].2;
	P1_Pracovisko.COM_Festo.DS1_1_Port0_IN[0].3;
	P1_Pracovisko.COM_Festo.DS1_1_Port0_IN[0].4;
	P1_Pracovisko.COM_Festo.DS1_1_Port0_IN[0].5;
	P1_Robot.IN.KodGripra_Bit0:= P1_Pracovisko.COM_Festo.DS1_1_Port0_IN[0].6;
	P1_Robot.IN.KodGripra_Bit1:= P1_Pracovisko.COM_Festo.DS1_1_Port0_IN[0].7;

	P1_Pracovisko.COM_Festo.DS1_1_Port0_IN[1].0;
	P1_Pracovisko.COM_Festo.DS1_1_Port0_IN[1].1;
	P1_Pracovisko.COM_Festo.DS1_1_Port0_IN[1].2;
	P1_Pracovisko.COM_Festo.DS1_1_Port0_IN[1].3;
	P1_Pracovisko.COM_Festo.DS1_1_Port0_IN[1].4;
	P1_Pracovisko.COM_Festo.DS1_1_Port0_IN[1].5;
	P1_Pracovisko.COM_Festo.DS1_1_Port0_IN[1].6;
	P1_Pracovisko.COM_Festo.DS1_1_Port0_IN[1].7;

	//Outputs//
	P1_Pracovisko.COM_Festo.DS1_1_Port0_OUT[0].0;
	P1_Pracovisko.COM_Festo.DS1_1_Port0_OUT[0].1;
	P1_Pracovisko.COM_Festo.DS1_1_Port0_OUT[0].2;
	P1_Pracovisko.COM_Festo.DS1_1_Port0_OUT[0].3;
	P1_Pracovisko.COM_Festo.DS1_1_Port0_OUT[0].4;
	P1_Pracovisko.COM_Festo.DS1_1_Port0_OUT[0].5;
	P1_Pracovisko.COM_Festo.DS1_1_Port0_OUT[0].6;
	P1_Pracovisko.COM_Festo.DS1_1_Port0_OUT[0].7;

	P1_Pracovisko.COM_Festo.DS1_1_Port0_OUT[1].0;
	P1_Pracovisko.COM_Festo.DS1_1_Port0_OUT[1].1;
	P1_Pracovisko.COM_Festo.DS1_1_Port0_OUT[1].2;
	P1_Pracovisko.COM_Festo.DS1_1_Port0_OUT[1].3;
	P1_Pracovisko.COM_Festo.DS1_1_Port0_OUT[1].4;
	P1_Pracovisko.COM_Festo.DS1_1_Port0_OUT[1].5;
	P1_Pracovisko.COM_Festo.DS1_1_Port0_OUT[1].6;
	P1_Pracovisko.COM_Festo.DS1_1_Port0_OUT[1].7;

	//*************Modul DS 1.1 IO link Port 1 - Banner*********************//
	//Inputs//
	P1_Vytah.Banner.Mapping_IN[0]:= P1_Pracovisko.COM_Festo.DS1_1_Port1_IN[0];
	P1_Vytah.Banner.Mapping_IN[1]:= P1_Pracovisko.COM_Festo.DS1_1_Port1_IN[1];
	P1_Vytah.Banner.Mapping_IN[2]:= P1_Pracovisko.COM_Festo.DS1_1_Port1_IN[2];
	P1_Vytah.Banner.Mapping_IN[3]:= P1_Pracovisko.COM_Festo.DS1_1_Port1_IN[3];
	P1_Vytah.Banner.Mapping_IN[4]:= P1_Pracovisko.COM_Festo.DS1_1_Port1_IN[4];
	P1_Vytah.Banner.Mapping_IN[5]:= P1_Pracovisko.COM_Festo.DS1_1_Port1_IN[5];
	P1_Vytah.Banner.Mapping_IN[6]:= P1_Pracovisko.COM_Festo.DS1_1_Port1_IN[6];
	P1_Vytah.Banner.Mapping_IN[7]:= P1_Pracovisko.COM_Festo.DS1_1_Port1_IN[7];
	P1_Vytah.Banner.Mapping_IN[8]:= P1_Pracovisko.COM_Festo.DS1_1_Port1_IN[8];
	P1_Vytah.Banner.Mapping_IN[9]:= P1_Pracovisko.COM_Festo.DS1_1_Port1_IN[9];
	P1_Vytah.Banner.Mapping_IN[10]:= P1_Pracovisko.COM_Festo.DS1_1_Port1_IN[10];
	P1_Vytah.Banner.Mapping_IN[11]:= P1_Pracovisko.COM_Festo.DS1_1_Port1_IN[11];
	P1_Vytah.Banner.Mapping_IN[12]:= P1_Pracovisko.COM_Festo.DS1_1_Port1_IN[12];
	P1_Vytah.Banner.Mapping_IN[13]:= P1_Pracovisko.COM_Festo.DS1_1_Port1_IN[13];
	P1_Vytah.Banner.Mapping_IN[14]:= P1_Pracovisko.COM_Festo.DS1_1_Port1_IN[14];
	P1_Vytah.Banner.Mapping_IN[15]:= P1_Pracovisko.COM_Festo.DS1_1_Port1_IN[15];

	//Outputs//
	P1_Pracovisko.COM_Festo.DS1_1_Port1_OUT[0]:= P1_Vytah.Banner.Mapping_OUT[0];
	P1_Pracovisko.COM_Festo.DS1_1_Port1_OUT[1]:= P1_Vytah.Banner.Mapping_OUT[1];
	P1_Pracovisko.COM_Festo.DS1_1_Port1_OUT[2]:= P1_Vytah.Banner.Mapping_OUT[2];
	P1_Pracovisko.COM_Festo.DS1_1_Port1_OUT[3]:= P1_Vytah.Banner.Mapping_OUT[3];
	P1_Pracovisko.COM_Festo.DS1_1_Port1_OUT[4]:= P1_Vytah.Banner.Mapping_OUT[4];
	P1_Pracovisko.COM_Festo.DS1_1_Port1_OUT[5]:= P1_Vytah.Banner.Mapping_OUT[5];
	P1_Pracovisko.COM_Festo.DS1_1_Port1_OUT[6]:= P1_Vytah.Banner.Mapping_OUT[6];
	P1_Pracovisko.COM_Festo.DS1_1_Port1_OUT[7]:= P1_Vytah.Banner.Mapping_OUT[7];
	P1_Pracovisko.COM_Festo.DS1_1_Port1_OUT[8]:= P1_Vytah.Banner.Mapping_OUT[8];
	P1_Pracovisko.COM_Festo.DS1_1_Port1_OUT[9]:= P1_Vytah.Banner.Mapping_OUT[9];
	P1_Pracovisko.COM_Festo.DS1_1_Port1_OUT[10]:= P1_Vytah.Banner.Mapping_OUT[10];
	P1_Pracovisko.COM_Festo.DS1_1_Port1_OUT[11]:= P1_Vytah.Banner.Mapping_OUT[11];
	P1_Pracovisko.COM_Festo.DS1_1_Port1_OUT[12]:= P1_Vytah.Banner.Mapping_OUT[12];
	P1_Pracovisko.COM_Festo.DS1_1_Port1_OUT[13]:= P1_Vytah.Banner.Mapping_OUT[13];
	P1_Pracovisko.COM_Festo.DS1_1_Port1_OUT[14]:= P1_Vytah.Banner.Mapping_OUT[14];
	P1_Pracovisko.COM_Festo.DS1_1_Port1_OUT[15]:= P1_Vytah.Banner.Mapping_OUT[15];

	//********Modul DS 1.1 IO link Port 2 - RFID snímač paletky výťahu**************//
	//Inputs//
	P1_Vytah.RFID_hlava.Mapping_IN[0]:= P1_Pracovisko.COM_Festo.DS1_1_Port2_IN[0];
	P1_Vytah.RFID_hlava.Mapping_IN[1]:= P1_Pracovisko.COM_Festo.DS1_1_Port2_IN[1];
	P1_Vytah.RFID_hlava.Mapping_IN[2]:= P1_Pracovisko.COM_Festo.DS1_1_Port2_IN[2];
	P1_Vytah.RFID_hlava.Mapping_IN[3]:= P1_Pracovisko.COM_Festo.DS1_1_Port2_IN[3];
	P1_Vytah.RFID_hlava.Mapping_IN[4]:= P1_Pracovisko.COM_Festo.DS1_1_Port2_IN[4];
	P1_Vytah.RFID_hlava.Mapping_IN[5]:= P1_Pracovisko.COM_Festo.DS1_1_Port2_IN[5];
	P1_Vytah.RFID_hlava.Mapping_IN[6]:= P1_Pracovisko.COM_Festo.DS1_1_Port2_IN[6];
	P1_Vytah.RFID_hlava.Mapping_IN[7]:= P1_Pracovisko.COM_Festo.DS1_1_Port2_IN[7];

	//Outputs//
	P1_Pracovisko.COM_Festo.DS1_1_Port2_OUT[0]:= P1_Vytah.RFID_hlava.Mapping_OUT[0];
	P1_Pracovisko.COM_Festo.DS1_1_Port2_OUT[1]:= P1_Vytah.RFID_hlava.Mapping_OUT[1];
	P1_Pracovisko.COM_Festo.DS1_1_Port2_OUT[2]:= P1_Vytah.RFID_hlava.Mapping_OUT[2];
	P1_Pracovisko.COM_Festo.DS1_1_Port2_OUT[3]:= P1_Vytah.RFID_hlava.Mapping_OUT[3];
	P1_Pracovisko.COM_Festo.DS1_1_Port2_OUT[4]:= P1_Vytah.RFID_hlava.Mapping_OUT[4];
	P1_Pracovisko.COM_Festo.DS1_1_Port2_OUT[5]:= P1_Vytah.RFID_hlava.Mapping_OUT[5];
	P1_Pracovisko.COM_Festo.DS1_1_Port2_OUT[6]:= P1_Vytah.RFID_hlava.Mapping_OUT[6];
	P1_Pracovisko.COM_Festo.DS1_1_Port2_OUT[7]:= P1_Vytah.RFID_hlava.Mapping_OUT[7];

	//*******Modul DS 1.1 IO link Port 3 - RFID snímač paletky stoper skrutkovania**********//
	//Inputs//
	P1_StoperSrobovania.RFID_hlava.Mapping_IN[0]:= P1_Pracovisko.COM_Festo.DS1_1_Port3_IN[0];
	P1_StoperSrobovania.RFID_hlava.Mapping_IN[1]:= P1_Pracovisko.COM_Festo.DS1_1_Port3_IN[1];
	P1_StoperSrobovania.RFID_hlava.Mapping_IN[2]:= P1_Pracovisko.COM_Festo.DS1_1_Port3_IN[2];
	P1_StoperSrobovania.RFID_hlava.Mapping_IN[3]:= P1_Pracovisko.COM_Festo.DS1_1_Port3_IN[3];
	P1_StoperSrobovania.RFID_hlava.Mapping_IN[4]:= P1_Pracovisko.COM_Festo.DS1_1_Port3_IN[4];
	P1_StoperSrobovania.RFID_hlava.Mapping_IN[5]:= P1_Pracovisko.COM_Festo.DS1_1_Port3_IN[5];
	P1_StoperSrobovania.RFID_hlava.Mapping_IN[6]:= P1_Pracovisko.COM_Festo.DS1_1_Port3_IN[6];
	P1_StoperSrobovania.RFID_hlava.Mapping_IN[7]:= P1_Pracovisko.COM_Festo.DS1_1_Port3_IN[7];

	//Outputs//
	P1_Pracovisko.COM_Festo.DS1_1_Port3_OUT[0]:= P1_StoperSrobovania.RFID_hlava.Mapping_OUT[0];
	P1_Pracovisko.COM_Festo.DS1_1_Port3_OUT[1]:= P1_StoperSrobovania.RFID_hlava.Mapping_OUT[1];
	P1_Pracovisko.COM_Festo.DS1_1_Port3_OUT[2]:= P1_StoperSrobovania.RFID_hlava.Mapping_OUT[2];
	P1_Pracovisko.COM_Festo.DS1_1_Port3_OUT[3]:= P1_StoperSrobovania.RFID_hlava.Mapping_OUT[3];
	P1_Pracovisko.COM_Festo.DS1_1_Port3_OUT[4]:= P1_StoperSrobovania.RFID_hlava.Mapping_OUT[4];
	P1_Pracovisko.COM_Festo.DS1_1_Port3_OUT[5]:= P1_StoperSrobovania.RFID_hlava.Mapping_OUT[5];
	P1_Pracovisko.COM_Festo.DS1_1_Port3_OUT[6]:= P1_StoperSrobovania.RFID_hlava.Mapping_OUT[6];
	P1_Pracovisko.COM_Festo.DS1_1_Port3_OUT[7]:= P1_StoperSrobovania.RFID_hlava.Mapping_OUT[7];

	//*********Modul DS 1.2 IO link Port 0 - Snímač vysunutia skrutkovačky K30****************//
	//Inputs//
	Convert_0.IN_Byte1:= P1_Pracovisko.COM_Festo.DS1_2_Port0_IN[0];
	Convert_0.IN_Byte0:= P1_Pracovisko.COM_Festo.DS1_2_Port0_IN[1];

	P1_Srobovanie.PAR.Skrutkov_K30_AktualHodnVysunutia:= Convert_0.OUT_UINT;
	Convert_0();

	//************************************Ventilový terminál*******************************************//

	//0-7
	P1_Pracovisko.COM_VentilovyTerminal[0].0 :=P1_Robot.OUT.Vakum_OFF;
	P1_Pracovisko.COM_VentilovyTerminal[0].1 :=P1_Robot.OUT.Vakum_ON;
	P1_Pracovisko.COM_VentilovyTerminal[0].2 :=P1_Srobovanie.OUT.Skrutkovacka_M5_Prisavanie_ON;
	P1_Pracovisko.COM_VentilovyTerminal[0].3 :=P1_Srobovanie.OUT.Skrutkovacka_M5_Prisavanie_OFF;
	P1_Pracovisko.COM_VentilovyTerminal[0].4 :=P1_Srobovanie.OUT.Skrutkovacka_M5_Odvzdusn_ON;
	P1_Pracovisko.COM_VentilovyTerminal[0].5 :=P1_Srobovanie.OUT.Skrutkovacka_M4_Odvzdusn_ON;
	P1_Pracovisko.COM_VentilovyTerminal[0].6 :=P1_Srobovanie.OUT.Skrutkovacka_M4_Prisavanie_ON;
	P1_Pracovisko.COM_VentilovyTerminal[0].7 :=P1_Srobovanie.OUT.Skrutkovacka_M4_Prisavanie_OFF;

	//8-15
	P1_Pracovisko.COM_VentilovyTerminal[1].0 :=P1_StoperSrobovania.OUT.ZasunStoper;
	P1_Pracovisko.COM_VentilovyTerminal[1].1 :=P1_AkumulacnyStoper.OUT.ZasunStoper;
	P1_Pracovisko.COM_VentilovyTerminal[1].2 :=P1_SpodnyStoper.OUT.ZasunStoper;
	P1_Pracovisko.COM_VentilovyTerminal[1].3;
	P1_Pracovisko.COM_VentilovyTerminal[1].4 :=P1_Srobovanie.SkrutSet_M4.OUT.ZhadzovaciVzduch_RUN;
	P1_Pracovisko.COM_VentilovyTerminal[1].5 :=P1_Srobovanie.SkrutSet_M4.OUT.TriediaciVzduch_RUN;
	P1_Pracovisko.COM_VentilovyTerminal[1].6 :=P1_Srobovanie.SkrutSet_M4.OUT.OtocPodavac_NaVstup;
	P1_Pracovisko.COM_VentilovyTerminal[1].7 :=P1_Srobovanie.SkrutSet_M4.OUT.OtocPodavac_NaVystup;

	//16-23
	P1_Pracovisko.COM_VentilovyTerminal[2].0 :=P1_Srobovanie.SkrutSet_K30.OUT.VibracnyHrniec.PrerusenieZasobovaniaSkrutiek;  (*SkrutkSet_K30.OUT.ZhadzovaciVzduch_RUN*)
	P1_Pracovisko.COM_VentilovyTerminal[2].1 :=P1_Srobovanie.SkrutSet_K30.OUT.VibracnyHrniec.TiedenieSkrutiek;                (*SkrutkSet_K30.OUT.TriediaciVzduch_RUN*)
	P1_Pracovisko.COM_VentilovyTerminal[2].2 :=P1_Srobovanie.SkrutSet_K30.OUT.VibracnyHrniec.OddelovacVysunut;                  (*SkrutkSet_K30.OUT.OddelovacSkrutiek_VYSUN *)
	P1_Pracovisko.COM_VentilovyTerminal[2].3 ;
	P1_Pracovisko.COM_VentilovyTerminal[2].4 :=P1_Srobovanie.SkrutSet_K30.OUT.VibracnyHrniec.VzduchNastreleniaSkrutky;         (*SkrutkSet_K30.OUT.NastrelSkrutkuDoBrzdy*)
	P1_Pracovisko.COM_VentilovyTerminal[2].5;
	P1_Pracovisko.COM_VentilovyTerminal[2].6 :=P1_Srobovanie.OUT.Skrutkovacka_K30_Prisavanie_ON;
	P1_Pracovisko.COM_VentilovyTerminal[2].7 :=P1_Srobovanie.OUT.Skrutkovacka_K30_Odvzdusn_ON;

	//24-31
	P1_Pracovisko.COM_VentilovyTerminal[3].0:=P1_Srobovanie.SkrutSet_K30.OUT.Brzda.PodajSkrutku; //Vysuň brzdu                 (*SkrutkSet_K30.OUT.Brzdu_VYSUN*)
	P1_Pracovisko.COM_VentilovyTerminal[3].1:=P1_Srobovanie.SkrutSet_K30.OUT.Brzda.ZakladnaPoloha; //Zasun brzdu                (*SkrutkSet_K30.OUT.Brzdu_ZASUN*)
	P1_Pracovisko.COM_VentilovyTerminal[3].2:=P1_Srobovanie.SkrutSet_K30.OUT.Brzda.OdsavanieNecistot;							(*SkrutkSet_K30.OUT.OdsavanieBrzdy_RUN*)
	P1_Pracovisko.COM_VentilovyTerminal[3].3:=P1_Srobovanie.SkrutSet_K30.OUT.Brzda.NastrelenieSkrutky;                  		(*SkrutkSet_K30.OUT.NastrelSkrutkuDoSkrutkovacky*)
	P1_Pracovisko.COM_VentilovyTerminal[3].4:=P1_Srobovanie.SkrutSet_M5.OUT.ZhadzovaciVzduch_RUN;
	P1_Pracovisko.COM_VentilovyTerminal[3].5:=P1_Srobovanie.SkrutSet_M5.OUT.TriediaciVzduch_RUN;
	P1_Pracovisko.COM_VentilovyTerminal[3].6:=P1_Srobovanie.SkrutSet_M5.OUT.OtocPodavac_NaVstup;
	P1_Pracovisko.COM_VentilovyTerminal[3].7:=P1_Srobovanie.SkrutSet_M5.OUT.OtocPodavac_NaVystup;

	//32-39
	P1_Pracovisko.COM_VentilovyTerminal[4].0 :=P1_Robot.OUT.OdistiGriper;
	P1_Pracovisko.COM_VentilovyTerminal[4].1 :=P1_Robot.OUT.ZaistiGriper;
	P1_Pracovisko.COM_VentilovyTerminal[4].2;
	P1_Pracovisko.COM_VentilovyTerminal[4].3;
	P1_Pracovisko.COM_VentilovyTerminal[4].4;
	P1_Pracovisko.COM_VentilovyTerminal[4].5;
	P1_Pracovisko.COM_VentilovyTerminal[4].6;
	P1_Pracovisko.COM_VentilovyTerminal[4].7;

	IF P1_Robot.OUT.OdistiGriper THEN
		P1_Pracovisko.COM_VentilovyTerminal[4].2:= FALSE;
		P1_Pracovisko.COM_VentilovyTerminal[4].3:= FALSE;
	ELSIF P1_Robot.OUT.Griper_OTVOR AND P1_Robot.IN.TypGripra_45F THEN
		P1_Pracovisko.COM_VentilovyTerminal[4].2:= TRUE;
		P1_Pracovisko.COM_VentilovyTerminal[4].3:= FALSE;
	ELSIF P1_Robot.OUT.Griper_ZATVOR AND P1_Robot.IN.TypGripra_45F THEN
		P1_Pracovisko.COM_VentilovyTerminal[4].2:= FALSE;
		P1_Pracovisko.COM_VentilovyTerminal[4].3:= TRUE;
	END_IF

	//40-47
	P1_Pracovisko.COM_VentilovyTerminal[5].0:=P1_Srobovanie.OUT.Skrutkovacku_K30_VYSUN;
	P1_Pracovisko.COM_VentilovyTerminal[5].1;
	P1_Pracovisko.COM_VentilovyTerminal[5].2:=P1_StoperSrobovania.OUT.Centrovanie_VYSUN;
	P1_Pracovisko.COM_VentilovyTerminal[5].3:=P1_StoperSrobovania.OUT.Centrovanie_ZASUN;
	P1_Pracovisko.COM_VentilovyTerminal[5].4;
	P1_Pracovisko.COM_VentilovyTerminal[5].5;
	P1_Pracovisko.COM_VentilovyTerminal[5].6;
	P1_Pracovisko.COM_VentilovyTerminal[5].7;

	//Limitné snímače serva zdvihu výťahu//
	P1_Vytah.IN.Zdvih_HornyLimSnimac:= P1_Vytah.ServoZdvihuVytahu.IN.PositiveLimitSwitch_Bit9;
	P1_Vytah.IN.Zdvih_SpodnyLimSnimac:= P1_Vytah.ServoZdvihuVytahu.IN.NegativeLimitSwitch_Bit8;

	//Volanie knižnic//
	P1_Vytah.ServoZdvihuVytahu();
	P1_Srobovanie.SkrutSet_K30();
	P1_Srobovanie.SkrutSet_M4();
	P1_Srobovanie.SkrutSet_M5();
	P1_Srobovanie.ServoManipulOsX();
	P1_Srobovanie.ServoManipulOsY();
	P1_Srobovanie.ServoManipulOsZ_M4();
	P1_Srobovanie.ServoManipulOsZ_M5();

END_PROGRAM

PROGRAM _EXIT
	(* Insert code here *)

END_PROGRAM
```

#### Variables.var - Local variables
```iecst
VAR
	Convert_0 : UsintToUint := (0);
END_VAR
```

### Program Logical/Program/Pracovisko_2/P2_Main (IEC)

#### Main.st - Init, cyclic, exit code
```iecst
PROGRAM _INIT
	(* Insert code here *)

END_PROGRAM

PROGRAM _CYCLIC

	//Volanie podprogramov//
	ProfinetKomunikaciaKAM1;
	ProfinetKomunikaciaKAM7;
	ProfinetKomunikaciaKAM8;
	ProfinetKomunikaciaKAM9;
	ProfinetKomunikaciaKAM10;
	ProfinetKomunikaciaKAM11;
	ProfinetKomunikaciaKAM12;
	ProfinetKomunikaciaKAM17;

	//**************************************Ukončenie cyklu pracoviska****************************************************//
	IF P2_Pracovisko.KoniecCyklu THEN
		IF P2_Dopravniky.Automat THEN
			P2_Dopravniky.KoniecCyklu:= TRUE;
		END_IF
		IF P2_SpodnyStoper.Automat THEN
			P2_SpodnyStoper.KoniecCyklu:= TRUE;
		END_IF
		IF P2_StoperZaklTesnenia.Automat THEN
			P2_StoperZaklTesnenia.KoniecCyklu:= TRUE;
		END_IF
		IF P2_ZakladacTesnenia.Automat THEN
			P2_ZakladacTesnenia.KoniecCyklu:= TRUE;
		END_IF
		IF P2_StoperMaticovacky.Automat THEN
			P2_StoperMaticovacky.KoniecCyklu:= TRUE;
		END_IF
		IF P2_AkumulacnyStoper.Automat THEN
			P2_AkumulacnyStoper.KoniecCyklu:= TRUE;
		END_IF
		IF P2_StoperSrobovania.Automat THEN
			P2_StoperSrobovania.KoniecCyklu:= TRUE;
		END_IF
		IF P2_Srobovanie.Automat THEN
			P2_Srobovanie.KoniecCyklu:= TRUE;
		END_IF
		IF P2_Robot.Automat THEN
			P2_Robot.KoniecCyklu:= TRUE;
		END_IF
		IF P2_StoperZvarania.Automat THEN
			P2_StoperZvarania.KoniecCyklu:= TRUE;
		END_IF
		IF P2_Zvaranie.Automat THEN
			P2_Zvaranie.KoniecCyklu:= TRUE;
		END_IF
		IF P2_Cistenie.Automat THEN
			P2_Cistenie.KoniecCyklu:= TRUE;
		END_IF
		P2_Pracovisko.KoniecCyklu:= FALSE;
	END_IF

	//************************************Ukončenie cyklu pri poruche*****************************************//
	//ST1 - Zakladanie tesnenia//
	IF P2_Pracovisko.STAV.Porucha_ST1 THEN
		IF P2_ZakladacTesnenia.Automat THEN
			P2_ZakladacTesnenia.Reset:= TRUE;
		END_IF
		IF P2_StoperZaklTesnenia.Automat THEN
			P2_StoperZaklTesnenia.Reset:= TRUE;
		END_IF
	END_IF

	//ST2 - Skrutkovanie matice//
	IF P2_Pracovisko.STAV.Porucha_ST2 THEN
		IF P2_Dopravniky.Automat THEN
			P2_Dopravniky.KoniecCyklu:= TRUE;
		END_IF
		IF P2_SpodnyStoper.Automat THEN
			P2_SpodnyStoper.KoniecCyklu:= TRUE;
		END_IF
		IF P2_AkumulacnyStoper.Automat THEN
			P2_AkumulacnyStoper.KoniecCyklu:= TRUE;
		END_IF
		IF P2_StoperSrobovania.Automat THEN
			P2_StoperSrobovania.KoniecCyklu:= TRUE;
		END_IF
		IF P2_Srobovanie.Automat THEN
			P2_Srobovanie.KoniecCyklu:= TRUE;
		END_IF
		IF P2_Robot.Automat THEN
			P2_Robot.KoniecCyklu:= TRUE;
		END_IF
		IF P2_StoperZvarania.Automat THEN
			P2_StoperZvarania.KoniecCyklu:= TRUE;
		END_IF
		IF P2_Zvaranie.Automat THEN
			P2_Zvaranie.KoniecCyklu:= TRUE;
		END_IF
		IF P2_Cistenie.Automat THEN
			P2_Cistenie.KoniecCyklu:= TRUE;
		END_IF
	END_IF

	//ST3 - Akumulačný stoper//
	IF P2_Pracovisko.STAV.Porucha_ST3 THEN
		IF P2_Dopravniky.Automat THEN
			P2_Dopravniky.KoniecCyklu:= TRUE;
		END_IF
		IF P2_SpodnyStoper.Automat THEN
			P2_SpodnyStoper.KoniecCyklu:= TRUE;
		END_IF
		IF P2_StoperMaticovacky.Automat THEN
			P2_StoperMaticovacky.KoniecCyklu:= TRUE;
		END_IF
		IF P2_AkumulacnyStoper.Automat THEN
			P2_AkumulacnyStoper.Reset:= TRUE;
		END_IF
		IF P2_StoperSrobovania.Automat THEN
			P2_StoperSrobovania.KoniecCyklu:= TRUE;
		END_IF
		IF P2_Srobovanie.Automat THEN
			P2_Srobovanie.KoniecCyklu:= TRUE;
		END_IF
		IF P2_Robot.Automat THEN
			P2_Robot.KoniecCyklu:= TRUE;
		END_IF
		IF P2_StoperZvarania.Automat THEN
			P2_StoperZvarania.KoniecCyklu:= TRUE;
		END_IF
		IF P2_Zvaranie.Automat THEN
			P2_Zvaranie.KoniecCyklu:= TRUE;
		END_IF
		IF P2_Cistenie.Automat THEN
			P2_Cistenie.KoniecCyklu:= TRUE;
		END_IF
	END_IF

	//ST4 - Šrobovanie//
	IF P2_Pracovisko.STAV.Porucha_ST4 THEN
		IF P2_Dopravniky.Automat THEN
			P2_Dopravniky.KoniecCyklu:= TRUE;
		END_IF
		IF P2_SpodnyStoper.Automat THEN
			P2_SpodnyStoper.KoniecCyklu:= TRUE;
		END_IF
		IF P2_StoperMaticovacky.Automat THEN
			P2_StoperMaticovacky.KoniecCyklu:= TRUE;
		END_IF
		IF P2_AkumulacnyStoper.Automat THEN
			P2_AkumulacnyStoper.KoniecCyklu:= TRUE;
		END_IF
		IF P2_Srobovanie.Automat THEN
			P2_Srobovanie.Reset:= TRUE;
		END_IF
		IF P2_Robot.Automat THEN
			P2_Robot.KoniecCyklu:= TRUE;
		END_IF
		IF P2_StoperZvarania.Automat THEN
			P2_StoperZvarania.KoniecCyklu:= TRUE;
		END_IF
		IF P2_Zvaranie.Automat THEN
			P2_Zvaranie.KoniecCyklu:= TRUE;
		END_IF
		IF P2_Cistenie.Automat THEN
			P2_Cistenie.KoniecCyklu:= TRUE;
		END_IF
	END_IF

	//ST5 - Zváranie a čistenie//
	IF P2_Pracovisko.STAV.Porucha_ST5 THEN
		IF P2_Dopravniky.Automat THEN
			P2_Dopravniky.KoniecCyklu:= TRUE;
		END_IF
		IF P2_SpodnyStoper.Automat THEN
			P2_SpodnyStoper.KoniecCyklu:= TRUE;
		END_IF
		IF P2_StoperMaticovacky.Automat THEN
			P2_StoperMaticovacky.KoniecCyklu:= TRUE;
		END_IF
		IF P2_AkumulacnyStoper.Automat THEN
			P2_AkumulacnyStoper.KoniecCyklu:= TRUE;
		END_IF
		IF P2_StoperSrobovania.Automat THEN
			P2_StoperSrobovania.KoniecCyklu:= TRUE;
		END_IF
		IF P2_Srobovanie.Automat THEN
			P2_Srobovanie.KoniecCyklu:= TRUE;
		END_IF
		IF P2_Robot.Automat THEN
			P2_Robot.KoniecCyklu:= TRUE;
		END_IF
		IF P2_Zvaranie.Automat THEN
			P2_Zvaranie.Reset:= TRUE;
		END_IF
		IF P2_Cistenie.Automat THEN
			P2_Cistenie.Reset:= TRUE;
		END_IF
	END_IF

	//*********************************Status prebieha ukončenie cyklu********************************************//
	IF P2_Dopravniky.KoniecCyklu OR
		P2_SpodnyStoper.KoniecCyklu OR
		P2_StoperZaklTesnenia.KoniecCyklu OR
		P2_ZakladacTesnenia.KoniecCyklu OR
		P2_StoperMaticovacky.KoniecCyklu OR
		P2_AkumulacnyStoper.KoniecCyklu OR
		P2_StoperSrobovania.KoniecCyklu OR
		P2_Srobovanie.KoniecCyklu OR
		P2_Robot.KoniecCyklu OR
		P2_StoperZvarania.KoniecCyklu OR
		P2_Zvaranie.KoniecCyklu OR
		P2_Cistenie.KoniecCyklu THEN
		P2_Pracovisko.STAV.UkoncenieCyklu_BUSY:= TRUE;
	ELSE
		P2_Pracovisko.STAV.UkoncenieCyklu_BUSY:= FALSE;
	END_IF

	//*******************************Resetovanie pracoviska po stlačení tlačítka Automat******************************************//
	IF P2_Vizu.TL_RezimAutomat THEN
		IF P2_Pracovisko.STAV.Manual THEN
			P2_Pracovisko.Reset:= TRUE;
		END_IF
		P2_Vizu.TL_RezimAutomat:= FALSE;
	END_IF

	//******************************************Resetovanie pracoviska************************************************************//
	IF P2_Pracovisko.Reset THEN
		P2_Dopravniky.Reset:= TRUE;
		P2_SpodnyStoper.Reset:= TRUE;
		P2_StoperZaklTesnenia.Reset:= TRUE;
		P2_ZakladacTesnenia.Reset:= TRUE;
		P2_StoperMaticovacky.Reset:= TRUE;
		P2_AkumulacnyStoper.Reset:= TRUE;
		P2_StoperSrobovania.Reset:= TRUE;
		P2_Srobovanie.Reset:= TRUE;
		P2_Robot.Reset:= TRUE;
		P2_StoperZvarania.Reset:= TRUE;
		P2_Zvaranie.Reset:= TRUE;
		P2_Cistenie.Reset:= TRUE;
		P2_Pracovisko.STAV.Porucha_ST1:= FALSE;
		P2_Pracovisko.STAV.Porucha_ST2:= FALSE;
		P2_Pracovisko.STAV.Porucha_ST3:= FALSE;
		P2_Pracovisko.STAV.Porucha_ST4:= FALSE;
		P2_Pracovisko.STAV.Porucha_ST5:= FALSE;
		P2_Pracovisko.Reset:= FALSE;
	END_IF

	//Prepnutie pracoviska do manualneho režimu//
	IF P2_Pracovisko.Manual THEN
		P2_Dopravniky.Manual:= TRUE;
		P2_SpodnyStoper.Manual:= TRUE;
		P2_StoperZaklTesnenia.Manual:= TRUE;
		P2_ZakladacTesnenia.Manual:= TRUE;
		P2_StoperMaticovacky.Manual:= TRUE;
		P2_AkumulacnyStoper.Manual:= TRUE;
		P2_StoperSrobovania.Manual:= TRUE;
		P2_Srobovanie.Manual:= TRUE;
		P2_Robot.Manual:= TRUE;
		P2_StoperZvarania.Manual:= TRUE;
		P2_Zvaranie.Manual:= TRUE;
		P2_Cistenie.Manual:= TRUE;
		P2_Pracovisko.Manual:= FALSE;
	END_IF

	//Spustenie pracoviska v automatickom režime//
	IF P2_Pracovisko.Automat THEN
		IF P2_Pracovisko.STAV.HardwareZaklTesnenia_OK THEN
			P2_StoperZaklTesnenia.Automat:= TRUE;
			P2_ZakladacTesnenia.Automat:= TRUE;
		END_IF
		IF Safety.STAV.P2_ZonaBunky_AKTIVNA AND P2_Pracovisko.STAV.HardwareBunky_OK THEN
			P2_Dopravniky.Automat:= TRUE;
			P2_SpodnyStoper.Automat:= TRUE;
			P2_StoperMaticovacky.Automat:= TRUE;
			P2_AkumulacnyStoper.Automat:= TRUE;
			P2_StoperSrobovania.Automat:= TRUE;
			P2_Srobovanie.Automat:= TRUE;
			P2_Robot.Automat:= TRUE;
			P2_StoperZvarania.Automat:= TRUE;
			P2_Zvaranie.Automat:= TRUE;
			P2_Cistenie.Automat:= TRUE;
		END_IF
		P2_Pracovisko.Automat:= FALSE;
	END_IF

	//***************************************************Príznaky pracoviska******************************************************//
	//Príznak pracovisko stav AUTOMAT//
	IF P2_Dopravniky.Automat OR
		P2_SpodnyStoper.Automat OR
		P2_StoperZaklTesnenia.Automat OR
		P2_ZakladacTesnenia.Automat OR
		P2_StoperMaticovacky.Automat OR
		P2_AkumulacnyStoper.Automat OR
		P2_StoperSrobovania.Automat OR
		P2_Srobovanie.Automat OR
		P2_Robot.Automat OR
		P2_StoperZvarania.Automat OR
		P2_Zvaranie.Automat OR
		P2_Cistenie.Automat THEN
		P2_Pracovisko.STAV.Automat:= TRUE;
	ELSE
		P2_Pracovisko.STAV.Automat:= FALSE;
	END_IF

	//Priznak pracovisko stav MANUAL//
	IF P2_Dopravniky.Manual OR
		P2_SpodnyStoper.Manual OR
		P2_StoperZaklTesnenia.Manual OR
		P2_ZakladacTesnenia.Manual OR
		P2_StoperMaticovacky.Manual OR
		P2_AkumulacnyStoper.Manual OR
		P2_StoperSrobovania.Manual OR
		P2_Srobovanie.Manual OR
		P2_Robot.Manual OR
		P2_StoperZvarania.Manual OR
		P2_Zvaranie.Manual OR
		P2_Cistenie.Manual THEN
		P2_Pracovisko.STAV.Manual:= TRUE;
	ELSE
		P2_Pracovisko.STAV.Manual:= FALSE;
	END_IF

	//Príznak pracovisko stav PoINIT//
	IF P2_Dopravniky.STAV.PoINIT AND
		P2_SpodnyStoper.STAV.PoINIT AND
		(P2_StoperZaklTesnenia.STAV.PoINIT OR NOT P2_StoperZaklTesnenia.Automat) AND
		(P2_ZakladacTesnenia.STAV.PoINIT OR NOT P2_ZakladacTesnenia.Automat) AND
		P2_Robot.STAV.PoINIT AND
		P2_StoperMaticovacky.STAV.PoINIT AND
		P2_AkumulacnyStoper.STAV.PoINIT AND
		P2_StoperSrobovania.STAV.PoINIT AND
		P2_Srobovanie.STAV.PoINIT AND
		P2_StoperZvarania.STAV.PoINIT AND
		P2_Zvaranie.STAV.PoINIT AND
		P2_Cistenie.STAV.PoINIT THEN
		P2_Pracovisko.STAV.PoINIT:= TRUE;
	ELSE
		P2_Pracovisko.STAV.PoINIT:= FALSE;
	END_IF

	//Príznak pracovisko stav READY//
	IF SC_P2_Dopravniky.Step = 1 AND
		SC_P2_SpodnyStoper.Step = 1 AND
		SC_P2_StoperZaklTesnenia.Step = 1 AND
		SC_P2_ZakladacTesnenia.Step = 1 AND
		SC_P2_StoperMaticovacky.Step = 1 AND
		SC_P2_AkumulacnyStoper.Step = 1 AND
		SC_P2_StoperSrobovania.Step = 1 AND
		SC_P2_Srobovanie.Step = 1 AND
		SC_P2_Robot.Step = 1 AND
		SC_P2_StoperZvarania.Step = 1 AND
		SC_P2_Zvaranie.Step = 1 AND
		SC_P2_Cistenie.Step = 1	THEN
		P2_Pracovisko.STAV.READY:= TRUE;
	ELSE
		P2_Pracovisko.STAV.READY:= FALSE;
	END_IF

	//Príznak pracovisko stav PORUCHA//
	IF P2_Pracovisko.STAV.Porucha_ST1 OR
		P2_Pracovisko.STAV.Porucha_ST2 OR
		P2_Pracovisko.STAV.Porucha_ST3 OR
		P2_Pracovisko.STAV.Porucha_ST4 OR
		P2_Pracovisko.STAV.Porucha_ST5 THEN
		P2_Pracovisko.STAV.PORUCHA:= TRUE;
	ELSE
		P2_Pracovisko.STAV.PORUCHA:= FALSE;
	END_IF

	//Príznak HW zakladača tesnenia OK//
	IF P2_Pracovisko.IN.TlakVzduchu_OK AND
		P2_Pracovisko.IN.ModulFesto_IO_KomOK AND
		P2_Pracovisko.IN.ModulWeidmuller_IO_KomOK AND
		P2_Pracovisko.IN.ServoZaklTesneniaPojazd_KomOK AND
		P2_Pracovisko.IN.ServoZaklTesneniaZdvih_KomOK AND
		(*P3_Pracovisko.IN.Kamery_ControlUnit_KomOK AND*)
		P2_Pracovisko.IN.VentilovyTerminal_KomOK THEN
		P2_Pracovisko.STAV.HardwareZaklTesnenia_OK:= TRUE;
	ELSE
		P2_Pracovisko.STAV.HardwareZaklTesnenia_OK:= FALSE;
	END_IF

	//Príznak HW Bunky OK//
	IF P2_Pracovisko.IN.TlakVzduchu_OK AND
		P2_Pracovisko.IN.ModulFesto_IO_KomOK AND
		P2_Pracovisko.IN.ModulWeidmuller_IO_KomOK AND
		P2_Pracovisko.IN.Robot_KomOK AND
		P2_Pracovisko.IN.Maticovacka_M4_KomOK AND
		P2_Pracovisko.IN.ServoManipulatorOsX_KomOK AND
		P2_Pracovisko.IN.ServoManipulatorOsY_KomOK AND
		P2_Pracovisko.IN.ServoManipulatorOsZ_M4_KomOK AND
		P2_Pracovisko.IN.ServoZvaraniaOsZ_KomOK AND
		P2_Pracovisko.IN.Skrutkovacka_M4_KomOK AND
		P2_Pracovisko.IN.Skrutkovacka_M5_KomOK AND
		P2_Pracovisko.IN.Skrutkovacka_M6_KomOK AND
		P2_Pracovisko.IN.VentilovyTerminal_KomOK AND
		P2_Srobovanie.IN.NapajanieSkrutkovackyM4_OK AND
		P2_Srobovanie.IN.NapajanieSkrutkovackyM5_OK AND
		P2_Srobovanie.IN.NapajanieSkrutkovackyM6_OK AND
		P2_Srobovanie.IN.NapajanieVibrolistyM4_OK AND
		P2_Srobovanie.IN.NapajanieZasobnikaM6_OK AND
		P2_Srobovanie.IN.NapajanieZasobnikaM4_OK AND
		P2_Pracovisko.IN.SmartKamera8_KomOK AND
		(*P3_Pracovisko.IN.Kamery_ControlUnit_KomOK AND*)
		P2_Pracovisko.IN.SmartKamera9_KomOK AND
		P2_Srobovanie.IN.NapajanieZasobnikaM5_OK THEN
		P2_Pracovisko.STAV.HardwareBunky_OK:= TRUE;
	ELSE
		P2_Pracovisko.STAV.HardwareBunky_OK:= FALSE;
	END_IF

	//Príznak skrutkovačky zasunuté//
	IF P2_Srobovanie.IN.Skrutkovacka_M5_ZASUNUTA AND P2_Srobovanie.IN.Skrutkovacka_M6_ZASUNUTA AND P2_Srobovanie.PAR.ManipulOsZ_M4_AktualnaPozicia < 5 THEN
		P2_Pracovisko.STAV.SkrutkovackyZasunute:= TRUE;
	ELSE
		P2_Pracovisko.STAV.SkrutkovackyZasunute:= FALSE;
	END_IF

	//*****************************Zapnutie osvetlenia pracoviska*********************************************************//
	P2_Pracovisko.OUT.OsvetlenieBunky_ON:= FALSE;
	P2_Pracovisko.OUT.OsvetleniePracZaklTesnenia_ON:= TRUE;
	P2_Pracovisko.OUT.Osvetlenie_CAM1_Svetlo1:= TRUE;
	P2_Pracovisko.OUT.Osvetlenie_CAM1_Svetlo2:= TRUE;
	P2_Pracovisko.OUT.Osvetlenie_CAM10:= TRUE;
	P2_Pracovisko.OUT.Osvetlenie_CAM11:= TRUE;
	P2_Pracovisko.OUT.Osvetlenie_CAM12:= TRUE;
	P2_Pracovisko.OUT.Srobovanie_OsvetleniePaletky_ON:= TRUE;
	P2_Pracovisko.OUT.Srobovanie_BodoveOsvetlenie_ON:= TRUE;

	//****************************************Ovládanie majáka***********************************************//
	//Zelené svetlo//

	IF P2_Pracovisko.STAV.Automat THEN
		P2_Pracovisko.OUT.Majak_ZeleneSvetlo_ON:= TRUE;
	ELSIF P2_Pracovisko.STAV.Manual THEN
		P2_Pracovisko.OUT.Majak_ZeleneSvetlo_ON:= Blikac500ms;
	ELSE
		P2_Pracovisko.OUT.Majak_ZeleneSvetlo_ON:= FALSE;
	END_IF

	//Oranžové svetlo//
	IF P2_Pracovisko.STAV.Automat AND NOT P2_Pracovisko.STAV.PoINIT THEN
		P2_Pracovisko.OUT.Majak_OranzoveSvetlo_ON:= TRUE;
	ELSE
		P2_Pracovisko.OUT.Majak_OranzoveSvetlo_ON:= FALSE;
	END_IF

	//Červené svetlo//
	IF NOT Safety.STAV.Linka_ZonaCS_AKTIVNA THEN
		P2_Pracovisko.OUT.Majak_CerveneSvetlo_ON:= TRUE;
	ELSIF P2_Pracovisko.STAV.Porucha_ST1 THEN
		P2_Pracovisko.OUT.Majak_CerveneSvetlo_ON:= TRUE;
	ELSIF P2_Pracovisko.STAV.Porucha_ST2 THEN
		P2_Pracovisko.OUT.Majak_CerveneSvetlo_ON:= TRUE;
	ELSIF P2_Pracovisko.STAV.Porucha_ST3 THEN
		P2_Pracovisko.OUT.Majak_CerveneSvetlo_ON:= TRUE;
	ELSIF P2_Pracovisko.STAV.Porucha_ST4 THEN
		P2_Pracovisko.OUT.Majak_CerveneSvetlo_ON:= TRUE;
	ELSIF P2_Pracovisko.STAV.Porucha_ST5 THEN
		P2_Pracovisko.OUT.Majak_CerveneSvetlo_ON:= TRUE;
	ELSE
		P2_Pracovisko.OUT.Majak_CerveneSvetlo_ON:= FALSE;
	END_IF

	//Zvuková signalizácia//
	//	IF EDGEPOS(P2_Pracovisko.STAV.Porucha_ST1) THEN
	//		P2_Pracovisko.OUT.Majak_Hukacka_ON:= Blikac500ms;
	//	ELSIF EDGEPOS(P2_Pracovisko.STAV.Porucha_ST2) THEN
	//		P2_Pracovisko.OUT.Majak_Hukacka_ON:= Blikac500ms;
	//	ELSIF EDGEPOS(P2_Pracovisko.STAV.Porucha_ST3) THEN
	//		P2_Pracovisko.OUT.Majak_Hukacka_ON:= Blikac500ms;
	//	ELSIF EDGEPOS(P2_Pracovisko.STAV.Porucha_ST4) THEN
	//		P2_Pracovisko.OUT.Majak_Hukacka_ON:= Blikac500ms;
	//	ELSIF EDGEPOS(P2_Pracovisko.STAV.Porucha_ST5) THEN
	//		P2_Pracovisko.OUT.Majak_Hukacka_ON:= Blikac500ms;
	//	END_IF
	//

END_PROGRAM

PROGRAM _EXIT
	(* Insert code here *)

END_PROGRAM
```

#### Variables.var - Local variables
```iecst
VAR
	Convert_0 : UsintToUint := (0);
	Convert_1 : UsintToUint := (0);
	Convert_2 : UsintToUint := (0);
	Convert_3 : UsintToUint := (0);
	Convert_4 : UsintToUint := (0);
	Convert_5 : UsintToUint := (0);
	Convert_6 : UsintToUint := (0);
	Convert_7 : UsintToUint := (0);
END_VAR
```

#### ProfinetKomunikaciaKAM7.st
```iecst
ACTION ProfinetKomunikaciaKAM7:
	//Control unit CAM5//

	//Vstupy pre kameru//
	CAM7.Profinet_PLC_OUTPUTS[0].3:= CAM7.CMD.Triger;

	//Výstupy z kamery//
	CAM7.STAV.READY:= CAM7.Profinet_PLC_INPUTS[0].0;
	CAM7.STAV.SWITCH:= CAM7.Profinet_PLC_INPUTS[0].1;
    CAM7.STAV.BUSY:= CAM7.Profinet_PLC_INPUTS[0].2;
    CAM7.STAV.Command_AKCEPTOVANY:= CAM7.Profinet_PLC_INPUTS[0].3;
    CAM7.STAV.Command_READY:= CAM7.Profinet_PLC_INPUTS[0].4;
    CAM7.STAV.Command_ERROR:= CAM7.Profinet_PLC_INPUTS[0].5;

	//Výsledky kamery//
	CAM7.RESULT.CitanieQRkodu_Filtra5H_OK:= CAM7.Profinet_PLC_INPUTS[2].0;

	//Prečítaný QR kód fitra 5H//
	IF EDGE(CAM7.STAV.SWITCH) THEN
		brsstrcpy(ADR(CAM7.RESULT.PrecitanyQRkod_Filtra5H),ADR(CAM7.Profinet_QRkod_Znaky));
	END_IF

	//Stav výsledky READY//
	IF EDGE(CAM7.STAV.SWITCH)THEN
		CAM7.STAV.Results_READY:= TRUE;
	END_IF

	//Run counter kamery//
	Convert_0.IN_Byte0:= CAM7.STAV.RunCounter_Byte1;
	Convert_0.IN_Byte1:= CAM7.STAV.RunCounter_Byte0;

	CAM7.STAV.RunCounter:= Convert_0.OUT_UINT;
	Convert_0();

END_ACTION
```

#### ProfinetKomunikaciaKAM8.st
```iecst
ACTION ProfinetKomunikaciaKAM8:
	//Smart kamera//

	CAM8.STAV.READY:= P2_Pracovisko.IN.SmartKamera8_KomOK;

	//Vstupy pre kameru//
	CAM8.Profinet_PLC_OUTPUTS[0].0:= CAM8.CMD.Triger;

	//Výstupy z kamery//
	CAM8.STAV.SWITCH:= CAM8.Profinet_PLC_INPUTS[12].0;

	//Výsledky kamery//
	CAM8.RESULT.PowerCP.CitanieQRkodu_PowerCP_OK:= CAM8.Profinet_PLC_INPUTS[0].0;

	//Prečítaný QR kód DPS//
	IF EDGE(CAM8.STAV.SWITCH) THEN
		brsstrcpy(ADR(CAM8.RESULT.PowerCP.PrecitanyQRkod_PowerCP),ADR(CAM8.Profinet_QRkod_Znaky));
	END_IF

	//Stav výsledky READY//
	IF EDGE(CAM8.STAV.SWITCH)THEN
		CAM8.STAV.Results_READY:= TRUE;
	END_IF

	//Run counter kamery//
	Convert_1.IN_Byte0:= CAM8.STAV.RunCounter_Byte1;
	Convert_1.IN_Byte1:= CAM8.STAV.RunCounter_Byte0;

	CAM8.STAV.RunCounter:= Convert_1.OUT_UINT;
	Convert_1();

END_ACTION
```

#### ProfinetKomunikaciaKAM9.st
```iecst
ACTION ProfinetKomunikaciaKAM9:
	//Smart kamera//

	CAM9.STAV.READY:= P2_Pracovisko.IN.SmartKamera9_KomOK;

	//Vstupy pre kameru//
	CAM9.Profinet_PLC_OUTPUTS[0].0:= CAM9.CMD.Triger;

	//Výstupy z kamery//
	CAM9.STAV.SWITCH:= CAM9.Profinet_PLC_INPUTS[12].0;

	//Výsledky kamery//
	CAM9.RESULT.PowerCP.PritomMatice:= CAM9.Profinet_PLC_INPUTS[0].0;
	CAM9.RESULT.PowerCP.PritomnBusbaru_5H:= CAM9.Profinet_PLC_INPUTS[0].1;

	//Stav výsledky READY//
	IF EDGE(CAM9.STAV.SWITCH)THEN
		CAM9.STAV.Results_READY:= TRUE;
		CAM9_PocetFotiek:= CAM9_PocetFotiek + 1;
	END_IF

	//Vymazanie adresára kamery//
	IF EDGEPOS(CAM9_PocetFotiek > 50) THEN
		FTP_CAM9.CMD.VymazFotku:= TRUE;
		FTP_CAM9.STATUS.VymazanieAdresaraKamery_BUSY:= TRUE;
	END_IF

	IF (FTP_CAM9.STATUS.KomunikaciaUkoncena OR FTP_CAM9.STATUS.KomunikaciaError) AND FTP_CAM9.STATUS.VymazanieAdresaraKamery_BUSY THEN
		FTP_CAM9.CMD.VymazFotku:= FALSE;
		FTP_CAM9.STATUS.VymazanieAdresaraKamery_BUSY:= FALSE;
	END_IF

	//Run counter kamery//
	Convert_2.IN_Byte0:= CAM9.STAV.RunCounter_Byte1;
	Convert_2.IN_Byte1:= CAM9.STAV.RunCounter_Byte0;

	CAM9.STAV.RunCounter:= Convert_2.OUT_UINT;
	Convert_2();

END_ACTION
```

#### ProfinetKomunikaciaKAM10.st
```iecst
ACTION ProfinetKomunikaciaKAM10:
	//Control Unit CAM 7//

	//Vstupy pre kameru//
	CAM10.Profinet_PLC_OUTPUTS[0].3:= CAM10.CMD.Triger;

	//Výstupy z kamery//
	CAM10.STAV.READY:= CAM10.Profinet_PLC_INPUTS[0].0;
	CAM10.STAV.SWITCH:= CAM10.Profinet_PLC_INPUTS[0].1;
    CAM10.STAV.BUSY:= CAM10.Profinet_PLC_INPUTS[0].2;
    CAM10.STAV.Command_AKCEPTOVANY:= CAM10.Profinet_PLC_INPUTS[0].3;
    CAM10.STAV.Command_READY:= CAM10.Profinet_PLC_INPUTS[0].4;
    CAM10.STAV.Command_ERROR:= CAM10.Profinet_PLC_INPUTS[0].5;

	//Výsledky kamery//
	CAM10.RESULT.Paletka.Pritomn_Busbarov_45F:= CAM10.Profinet_PLC_INPUTS[2].0;
	CAM10.RESULT.Paletka.Pritomn_Busbarov_5H:= CAM10.Profinet_PLC_INPUTS[2].1;
	CAM10.RESULT.Paletka.Pritomn_PowerCP_4F:= CAM10.Profinet_PLC_INPUTS[2].2;
	CAM10.RESULT.Paletka.Pritomn_PowerCP_5F:= CAM10.Profinet_PLC_INPUTS[2].3;
	CAM10.RESULT.Paletka.Pritomn_PowerCP_5H:= CAM10.Profinet_PLC_INPUTS[2].4;

	//Stav výsledky READY//
	IF EDGE(CAM10.STAV.SWITCH)THEN
		CAM10.STAV.Results_READY:= TRUE;
		CAM10_PocetFotiek:= CAM10_PocetFotiek + 1;
	END_IF

	//Vymazanie adresára kamery//
	IF EDGEPOS(CAM10_PocetFotiek > 50) THEN
		FTP_CAM10.CMD.VymazFotku:= TRUE;
		FTP_CAM10.STATUS.VymazanieAdresaraKamery_BUSY:= TRUE;
	END_IF

	IF (FTP_CAM10.STATUS.KomunikaciaUkoncena OR FTP_CAM10.STATUS.KomunikaciaError) AND FTP_CAM10.STATUS.VymazanieAdresaraKamery_BUSY THEN
		FTP_CAM10.CMD.VymazFotku:= FALSE;
		FTP_CAM10.STATUS.VymazanieAdresaraKamery_BUSY:= FALSE;
	END_IF

	//Run counter kamery//
	Convert_3.IN_Byte0:= CAM10.STAV.RunCounter_Byte1;
	Convert_3.IN_Byte1:= CAM10.STAV.RunCounter_Byte0;

	CAM10.STAV.RunCounter:= Convert_3.OUT_UINT;
	Convert_3();

END_ACTION
```

#### ProfinetKomunikaciaKAM11.st
```iecst
ACTION ProfinetKomunikaciaKAM11:

	//Control Unit CAM 8//

	//Vstupy pre kameru//
	CAM11.Profinet_PLC_OUTPUTS[0].3:= CAM11.CMD.Triger;

	//Výstupy z kamery//
	CAM11.STAV.READY:= CAM11.Profinet_PLC_INPUTS[0].0;
	CAM11.STAV.SWITCH:= CAM11.Profinet_PLC_INPUTS[0].1;
    CAM11.STAV.BUSY:= CAM11.Profinet_PLC_INPUTS[0].2;
    CAM11.STAV.Command_AKCEPTOVANY:= CAM11.Profinet_PLC_INPUTS[0].3;
    CAM11.STAV.Command_READY:= CAM11.Profinet_PLC_INPUTS[0].4;
    CAM11.STAV.Command_ERROR:= CAM11.Profinet_PLC_INPUTS[0].5;

	//Výsledky kamery//
	CAM11.RESULT.Paletka.Pritomn_PowerCP_4F:= CAM11.Profinet_PLC_INPUTS[2].0;
	CAM11.RESULT.Paletka.Pritomn_PowerCP_5F:= CAM11.Profinet_PLC_INPUTS[2].1;
	CAM11.RESULT.Paletka.Pritomn_PowerCP_5H:= CAM11.Profinet_PLC_INPUTS[2].2;
	CAM11.RESULT.PowerCP.Pritomn_LavyMVcase:= CAM11.Profinet_PLC_INPUTS[2].3;
	CAM11.RESULT.PowerCP.Pritomn_PravyMVcase:= CAM11.Profinet_PLC_INPUTS[2].4;
	CAM11.RESULT.PowerCP.LavyBusbar_Zvaranie_OK:= CAM11.Profinet_PLC_INPUTS[2].5;
	CAM11.RESULT.PowerCP.PravyBusbar_Zvaranie_OK:= CAM11.Profinet_PLC_INPUTS[2].6;
	CAM11.RESULT.PowerCP.Pritomn_TopCover_4F:= CAM11.Profinet_PLC_INPUTS[2].7;

	CAM11.RESULT.PowerCP.Pritomn_TopCover_5F:= CAM11.Profinet_PLC_INPUTS[3].0;
	CAM11.RESULT.PowerCP.Pritomn_TopCover_5H:= CAM11.Profinet_PLC_INPUTS[3].1;

	//Stav výsledky READY//
	IF EDGE(CAM11.STAV.SWITCH)THEN
		CAM11.STAV.Results_READY:= TRUE;
		CAM11_PocetFotiek:= CAM11_PocetFotiek + 1;
	END_IF

	//Vymazanie adresára kamery//
	IF EDGEPOS(CAM11_PocetFotiek > 50) THEN
		FTP_CAM11.CMD.VymazFotku:= TRUE;
		FTP_CAM11.STATUS.VymazanieAdresaraKamery_BUSY:= TRUE;
	END_IF

	IF (FTP_CAM11.STATUS.KomunikaciaUkoncena OR FTP_CAM11.STATUS.KomunikaciaError) AND FTP_CAM11.STATUS.VymazanieAdresaraKamery_BUSY THEN
		FTP_CAM11.CMD.VymazFotku:= FALSE;
		FTP_CAM11.STATUS.VymazanieAdresaraKamery_BUSY:= FALSE;
	END_IF

	//Run counter kamery//
	Convert_4.IN_Byte0:= CAM11.STAV.RunCounter_Byte1;
	Convert_4.IN_Byte1:= CAM11.STAV.RunCounter_Byte0;

	CAM11.STAV.RunCounter:= Convert_4.OUT_UINT;
	Convert_4();

END_ACTION
```

#### ProfinetKomunikaciaKAM12.st
```iecst
ACTION ProfinetKomunikaciaKAM12:
	//Control Unit CAM 9//

	//Vstupy pre kameru//
	CAM12.Profinet_PLC_OUTPUTS[0].3:= CAM12.CMD.Triger;

	//Výstupy z kamery//
	CAM12.STAV.READY:= CAM12.Profinet_PLC_INPUTS[0].0;
	CAM12.STAV.SWITCH:= CAM12.Profinet_PLC_INPUTS[0].1;
    CAM12.STAV.BUSY:= CAM12.Profinet_PLC_INPUTS[0].2;
    CAM12.STAV.Command_AKCEPTOVANY:= CAM12.Profinet_PLC_INPUTS[0].3;
    CAM12.STAV.Command_READY:= CAM12.Profinet_PLC_INPUTS[0].4;
    CAM12.STAV.Command_ERROR:= CAM12.Profinet_PLC_INPUTS[0].5;

	//Výsledky kamery//
	CAM12.RESULT.Paletka.Pritomn_TopCover_4F:= CAM12.Profinet_PLC_INPUTS[2].0;
	CAM12.RESULT.Paletka.Pritomn_TopCover_5F:= CAM12.Profinet_PLC_INPUTS[2].1;
	CAM12.RESULT.Paletka.Pritomn_TopCover_5H:= CAM12.Profinet_PLC_INPUTS[2].2;
	CAM12.RESULT.Paletka.Pritomn_PravyMVcase:= CAM12.Profinet_PLC_INPUTS[2].3;
	CAM12.RESULT.Paletka.Pritomn_LavyMVcase:= CAM12.Profinet_PLC_INPUTS[2].4;

	//Stav výsledky READY//
	IF EDGE(CAM12.STAV.SWITCH)THEN
		CAM12.STAV.Results_READY:= TRUE;
		CAM12_PocetFotiek:= CAM12_PocetFotiek + 1;
	END_IF

	//Vymazanie adresára kamery//
	IF EDGEPOS(CAM12_PocetFotiek > 50) THEN
		FTP_CAM12.CMD.VymazFotku:= TRUE;
		FTP_CAM12.STATUS.VymazanieAdresaraKamery_BUSY:= TRUE;
	END_IF

	IF (FTP_CAM12.STATUS.KomunikaciaUkoncena OR FTP_CAM12.STATUS.KomunikaciaError) AND FTP_CAM12.STATUS.VymazanieAdresaraKamery_BUSY THEN
		FTP_CAM12.CMD.VymazFotku:= FALSE;
		FTP_CAM12.STATUS.VymazanieAdresaraKamery_BUSY:= FALSE;
	END_IF

	//Run counter kamery//
	Convert_5.IN_Byte0:= CAM12.STAV.RunCounter_Byte1;
	Convert_5.IN_Byte1:= CAM12.STAV.RunCounter_Byte0;

	CAM12.STAV.RunCounter:= Convert_5.OUT_UINT;
	Convert_5();

END_ACTION
```

#### ProfinetKomunikaciaKAM17.st
```iecst
ACTION ProfinetKomunikaciaKAM17:
	//Control Unit CAM 6 //

	//Vstupy pre kameru//
	CAM17.Profinet_PLC_OUTPUTS[0].3:= CAM17.CMD.Triger;

	//Výstupy z kamery//
	CAM17.STAV.READY:= CAM17.Profinet_PLC_INPUTS[0].0;
	CAM17.STAV.SWITCH:= CAM17.Profinet_PLC_INPUTS[0].1;
    CAM17.STAV.BUSY:= CAM17.Profinet_PLC_INPUTS[0].2;
    CAM17.STAV.Command_AKCEPTOVANY:= CAM17.Profinet_PLC_INPUTS[0].3;
    CAM17.STAV.Command_READY:= CAM17.Profinet_PLC_INPUTS[0].4;
    CAM17.STAV.Command_ERROR:= CAM17.Profinet_PLC_INPUTS[0].5;

	//Výsledky kamery//
	CAM17.RESULT.Paletka.Pritomn_PowerCP_4F:= CAM17.Profinet_PLC_INPUTS[2].0;
	CAM17.RESULT.Paletka.Pritomn_PowerCP_5F:= CAM17.Profinet_PLC_INPUTS[2].1;
	CAM17.RESULT.Paletka.Pritomn_PowerCP_5H:= CAM17.Profinet_PLC_INPUTS[2].2;
	CAM17.RESULT.Paletka.PrazdnaPoziciaTopCoveru:= CAM17.Profinet_PLC_INPUTS[2].3;
	CAM17.RESULT.Paletka.Pritomn_TopCoveru_4F:= CAM17.Profinet_PLC_INPUTS[2].4;
	CAM17.RESULT.Paletka.Pritomn_TopCoveru_5F:= CAM17.Profinet_PLC_INPUTS[2].5;
	CAM17.RESULT.Paletka.Pritomn_TopCoveru_5H:= CAM17.Profinet_PLC_INPUTS[2].6;
	CAM17.RESULT.Paletka.Pritomn_Busbary_5H:= CAM17.Profinet_PLC_INPUTS[2].7;

	CAM17.RESULT.Paletka.Pritomn_Busbary_5F:= CAM17.Profinet_PLC_INPUTS[3].0;
	CAM17.RESULT.Paletka.Pritomn_Busbary_4F:= CAM17.Profinet_PLC_INPUTS[3].1;
	CAM17.RESULT.Paletka.Pritomn_LavyMVcase:= CAM17.Profinet_PLC_INPUTS[3].2;
	CAM17.RESULT.Paletka.Pritomn_PravyMVcase:= CAM17.Profinet_PLC_INPUTS[3].3;

	//Stav výsledky READY//
	IF EDGE(CAM17.STAV.SWITCH)THEN
		CAM17.STAV.Results_READY:= TRUE;
		CAM17_PocetFotiek:= CAM17_PocetFotiek + 1;
	END_IF

	//Vymazanie adresára kamery//
	IF EDGEPOS(CAM17_PocetFotiek > 50) THEN
		FTP_CAM17.CMD.VymazFotku:= TRUE;
		FTP_CAM17.STATUS.VymazanieAdresaraKamery_BUSY:= TRUE;
	END_IF

	IF (FTP_CAM17.STATUS.KomunikaciaUkoncena OR FTP_CAM17.STATUS.KomunikaciaError) AND FTP_CAM17.STATUS.VymazanieAdresaraKamery_BUSY THEN
		FTP_CAM17.CMD.VymazFotku:= FALSE;
		FTP_CAM17.STATUS.VymazanieAdresaraKamery_BUSY:= FALSE;
	END_IF

	//Run counter kamery//
	Convert_6.IN_Byte0:= CAM17.STAV.RunCounter_Byte1;
	Convert_6.IN_Byte1:= CAM17.STAV.RunCounter_Byte0;

	CAM17.STAV.RunCounter:= Convert_6.OUT_UINT;
	Convert_6();

END_ACTION
```

#### ProfinetKomunikaciaKAM1.st
```iecst
ACTION ProfinetKomunikaciaKAM1:
	//Control unit CAM4//

	//Vstupy pre kameru//
	CAM1.Profinet_PLC_OUTPUTS[0].3:= CAM1.CMD.Triger;

	//Výstupy z kamery//
	CAM1.STAV.READY:= CAM1.Profinet_PLC_INPUTS[0].0;
	CAM1.STAV.SWITCH:= CAM1.Profinet_PLC_INPUTS[0].1;
	CAM1.STAV.BUSY:= CAM1.Profinet_PLC_INPUTS[0].2;
	CAM1.STAV.Command_AKCEPTOVANY:= CAM1.Profinet_PLC_INPUTS[0].3;
	CAM1.STAV.Command_READY:= CAM1.Profinet_PLC_INPUTS[0].4;
	CAM1.STAV.Command_ERROR:= CAM1.Profinet_PLC_INPUTS[0].5;

	//Výsledky kamery//
	CAM1.RESULT.ZalozenieTesnenia_OK:= CAM1.Profinet_PLC_INPUTS[2].0;
	CAM1.RESULT.NepritomnostTesnenia:= CAM1.Profinet_PLC_INPUTS[2].1;

	///Stav výsledky READY//
	IF EDGE(CAM1.STAV.SWITCH)THEN
		CAM1.STAV.Results_READY:= TRUE;
		CAM1_PocetFotiek:= CAM1_PocetFotiek + 1;
	END_IF

	//Vymazanie adresára kamery//
	IF EDGEPOS(CAM1_PocetFotiek > 50) THEN
		FTP_CAM1.CMD.VymazFotku:= TRUE;
		FTP_CAM1.STATUS.VymazanieAdresaraKamery_BUSY:= TRUE;
	END_IF

	IF (FTP_CAM1.STATUS.KomunikaciaUkoncena OR FTP_CAM1.STATUS.KomunikaciaError) AND FTP_CAM1.STATUS.VymazanieAdresaraKamery_BUSY THEN
		FTP_CAM1.CMD.VymazFotku:= FALSE;
		FTP_CAM1.STATUS.VymazanieAdresaraKamery_BUSY:= FALSE;
	END_IF

	//Run counter kamery//
	Convert_7.IN_Byte0:= CAM1.STAV.RunCounter_Byte1;
	Convert_7.IN_Byte1:= CAM1.STAV.RunCounter_Byte0;

	CAM1.STAV.RunCounter:= Convert_7.OUT_UINT;
	Convert_7();

END_ACTION
```

### Program Logical/Program/Pracovisko_2/P2_Dopravniky (IEC)

#### Main.st - Init, cyclic, exit code
```iecst
PROGRAM _INIT
	(* Insert code here *)

END_PROGRAM

PROGRAM _CYCLIC

	//Volanie funkcie SequenceControl//
	SequenceControl(SC:= SC_P2_Dopravniky);

	//Reset sekcie //
	IF P2_Dopravniky.Reset THEN
		SC_P2_Dopravniky.Step:= 0;
		P2_Dopravniky.Reset:= FALSE;
	ELSIF NOT Safety.STAV.Linka_ZonaCS_AKTIVNA THEN
		SC_P2_Dopravniky.Step:= 0;
	END_IF

	CASE SC_P2_Dopravniky.Step OF

		0:
			SC_P2_Dopravniky.StepName:='0 - Nulovanie';
			P2_Dopravniky.Automat:= FALSE;
			P2_Dopravniky.KoniecCyklu:= FALSE;
			P2_Dopravniky.Manual:= FALSE;
			P2_Dopravniky.STAV.PoINIT:= FALSE;
			P2_Dopravniky.OUT.DopravnikBunky_ON:= FALSE;
			P2_Dopravniky.OUT.VratnyDopravnik_ON:= FALSE;

			IF Safety.STAV.Linka_ZonaCS_AKTIVNA AND P2_Pracovisko.STAV.HardwareBunky_OK AND NOT P2_Pracovisko.STAV.Porucha_ST2 AND NOT P2_Pracovisko.STAV.Porucha_ST3 AND NOT P2_Pracovisko.STAV.Porucha_ST4 AND NOT P2_Pracovisko.STAV.Porucha_ST5 THEN
				SC_P2_Dopravniky.ResetStep:= TRUE;
				SC_P2_Dopravniky.Step:= 1;
			END_IF

		1:
			SC_P2_Dopravniky.StepName:='1 - Cakam na spustenie vyroby';
			P2_Dopravniky.KoniecCyklu:= FALSE;
			IF P2_Dopravniky.Automat THEN
				SC_P2_Dopravniky.Step:= 2;
			ELSIF P2_Dopravniky.Manual THEN
				SC_P2_Dopravniky.Step:= 700;
			END_IF

			//********************************************************Inicializácia****************************************************************************//

		2:
			SC_P2_Dopravniky.StepName:='2 - Inicializacia - cakam na spustenie inicializacie';
			SC_P2_Dopravniky.IdleTime.PT:= T#1s;
			SC_P2_Dopravniky.AlarmTime.PT:= T#5s;

			IF P2_Pracovisko.STAV.SkrutkovackyZasunute AND P2_Robot.STAV.PoINIT THEN
				SC_P2_Dopravniky.IdleTime.IN:= TRUE;
			ELSE
				SC_P2_Dopravniky.IdleTime.IN:= FALSE;
			END_IF

			IF SC_P2_Dopravniky.IdleTime.Q THEN
				SC_P2_Dopravniky.ResetStep:= TRUE;
				SC_P2_Dopravniky.Step:= 3;
			END_IF

		3:
			SC_P2_Dopravniky.StepName:='3 - Inicializacia - inicializacia tlmenia stoprov';
			SC_P2_Dopravniky.IdleTime.PT:= T#1s;
			SC_P2_Dopravniky.AlarmTime.PT:= T#5s;

			IF P2_StoperZaklTesnenia.RFID_hlava.PritomnostPaletky AND
				P2_StoperMaticovacky.RFID_hlava.PritomnostPaletky AND
				P2_AkumulacnyStoper.IN.PritomnostPaletky AND
				P2_StoperSrobovania.RFID_hlava.PritomnostPaletky AND
				P2_StoperZvarania.RFID_hlava.PritomnostPaletky AND
				P2_SpodnyStoper.IN.PritomnostPaletky THEN
				SC_P2_Dopravniky.ResetStep:= TRUE;
				SC_P2_Dopravniky.Step:= 5;
			ELSE
				IF NOT P2_StoperZaklTesnenia.RFID_hlava.PritomnostPaletky THEN
					P2_StoperZaklTesnenia.OUT.ZasunStoper:= TRUE;
				END_IF
				IF NOT P2_StoperMaticovacky.RFID_hlava.PritomnostPaletky AND P2_StoperMaticovacky.IN.Centrovanie_ZASUNUTE THEN
					P2_StoperMaticovacky.OUT.ZasunStoper:= TRUE;
				END_IF
				IF NOT P2_AkumulacnyStoper.IN.PritomnostPaletky THEN
					P2_AkumulacnyStoper.OUT.ZasunStoper:= TRUE;
				END_IF
				IF NOT P2_StoperSrobovania.RFID_hlava.PritomnostPaletky AND P2_StoperSrobovania.IN.Centrovanie_ZASUNUTE THEN
					P2_StoperSrobovania.OUT.ZasunStoper:= TRUE;
				END_IF
				IF NOT P2_StoperZvarania.RFID_hlava.PritomnostPaletky AND P2_StoperZvarania.IN.Centrovanie_ZASUNUTE THEN
					P2_StoperZvarania.OUT.ZasunStoper:= TRUE;
				END_IF
				IF NOT P2_SpodnyStoper.IN.PritomnostPaletky THEN
					P2_SpodnyStoper.OUT.ZasunStoper:= TRUE;
				END_IF
				SC_P2_Dopravniky.IdleTime.IN:= TRUE;
			END_IF

			IF SC_P2_Dopravniky.IdleTime.Q THEN
				P2_StoperZaklTesnenia.OUT.ZasunStoper:= FALSE;
				P2_StoperMaticovacky.OUT.ZasunStoper:= FALSE;
				P2_AkumulacnyStoper.OUT.ZasunStoper:= FALSE;
				P2_StoperSrobovania.OUT.ZasunStoper:= FALSE;
				P2_StoperZvarania.OUT.ZasunStoper:= FALSE;
				P2_SpodnyStoper.OUT.ZasunStoper:= FALSE;
				SC_P2_Dopravniky.ResetStep:= TRUE;
				SC_P2_Dopravniky.Step:= 5;
			END_IF

		5:
			SC_P2_Dopravniky.StepName:='5 - Inicializacia - ukoncenie inicializacie';
			SC_P2_Dopravniky.IdleTime.PT:= T#5s;
			SC_P2_Dopravniky.AlarmTime.PT:= T#5s;

			P2_Dopravniky.OUT.DopravnikBunky_ON:= TRUE;
			P2_Dopravniky.OUT.VratnyDopravnik_ON:= TRUE;
			SC_P2_Dopravniky.IdleTime.IN:= TRUE;

			IF SC_P2_Dopravniky.IdleTime.Q THEN
				P2_Dopravniky.STAV.PoINIT:= TRUE;
				SC_P2_Dopravniky.ResetStep:= TRUE;
				SC_P2_Dopravniky.Step:= 100;
			END_IF

			//********************************************************Automatický režim****************************************************************************//

		100:
			SC_P2_Dopravniky.StepName:='100 - Automaticky Rezim - cakam na vypnutie dopravnikou';
			SC_P2_Dopravniky.IdleTime.PT:= T#200ms;
			SC_P2_Dopravniky.AlarmTime.PT:= T#5s;

			IF P2_Dopravniky.KoniecCyklu AND
				NOT P2_StoperZaklTesnenia.STAV.PrebiehaVyvezeniePaletky AND
				NOT P2_StoperMaticovacky.Automat AND
				NOT P2_AkumulacnyStoper.Automat AND
				NOT P2_StoperSrobovania.Automat AND
				NOT P2_StoperZvarania.Automat AND
				NOT P2_SpodnyStoper.Automat THEN
				SC_P2_Dopravniky.ResetStep:= TRUE;
				SC_P2_Dopravniky.Step:= 0;
			END_IF

			//*******************************************************Manuálny režim*******************************************************************************//
		700:
			SC_P2_Dopravniky.StepName:='700 - Manualny Rezim';
			SC_P2_Dopravniky.IdleTime.PT:= T#8s;
			SC_P2_Dopravniky.AlarmTime.PT:= T#5s;

	END_CASE

END_PROGRAM

PROGRAM _EXIT
	(* Insert code here *)

END_PROGRAM
```

### Program Logical/Program/Pracovisko_2/P2_SpodnyStoper (IEC)

#### Main.st - Init, cyclic, exit code
```iecst
PROGRAM _INIT
	(* Insert code here *)

END_PROGRAM

PROGRAM _CYCLIC

	//Volanie funkcie SequenceControl//
	SequenceControl(SC:= SC_P2_SpodnyStoper);

	//Reset sekcie //
	IF P2_SpodnyStoper.Reset THEN
		SC_P2_SpodnyStoper.Step:= 0;
		P2_SpodnyStoper.Reset:= FALSE;
	ELSIF NOT Safety.STAV.Linka_ZonaCS_AKTIVNA THEN
		SC_P2_SpodnyStoper.Step:= 0;
	END_IF

	CASE SC_P2_SpodnyStoper.Step OF

		0:
			SC_P2_SpodnyStoper.StepName:='0 - Nulovanie';
			P2_SpodnyStoper.Automat:= FALSE;
			P2_SpodnyStoper.KoniecCyklu:= FALSE;
			P2_SpodnyStoper.Manual:= FALSE;
			P2_SpodnyStoper.STAV.PoINIT:= FALSE;
			P2_SpodnyStoper.STAV.PrebiehaVyvezeniePaletky:= FALSE;
			P2_SpodnyStoper.OUT.ZasunStoper:= FALSE;

			IF Safety.STAV.Linka_ZonaCS_AKTIVNA AND Safety.STAV.P2_ZonaBunky_AKTIVNA AND P2_Pracovisko.STAV.HardwareBunky_OK THEN
				SC_P2_SpodnyStoper.ResetStep:= TRUE;
				SC_P2_SpodnyStoper.Step:= 1;
			END_IF

		1:
			SC_P2_SpodnyStoper.StepName:='1 - Cakam na spustenie vyroby';
			P2_SpodnyStoper.KoniecCyklu:= FALSE;
			IF P2_SpodnyStoper.Automat THEN
				SC_P2_SpodnyStoper.Step:= 2;
			ELSIF P2_SpodnyStoper.Manual THEN
				SC_P2_SpodnyStoper.Step:= 700;
			END_IF

			//********************************************************Inicializácia****************************************************************************//
		2:
			SC_P2_SpodnyStoper.StepName:='2 - Inicializacia - cakam na spustenie inicializacie';
			SC_P2_SpodnyStoper.IdleTime.PT:= T#4s;
			SC_P2_SpodnyStoper.AlarmTime.PT:= T#5s;

			IF P2_Dopravniky.STAV.PoINIT THEN
				SC_P2_SpodnyStoper.ResetStep:= TRUE;
				SC_P2_SpodnyStoper.Step:= 3;
			END_IF

		3:
			SC_P2_SpodnyStoper.StepName:='3 - Inicializacia - hladanie paletky';
			SC_P2_SpodnyStoper.IdleTime.PT:= T#5s;
			SC_P2_SpodnyStoper.AlarmTime.PT:= T#5s;
			SC_P2_SpodnyStoper.IdleTime.IN:= TRUE;

			IF P2_SpodnyStoper.IN.PritomnostPaletky THEN
				P2_SpodnyStoper.STAV.PoINIT:= TRUE;
				SC_P2_SpodnyStoper.ResetStep:= TRUE;
				SC_P2_SpodnyStoper.Step:= 101;
			ELSIF SC_P2_SpodnyStoper.IdleTime.Q THEN
				P2_SpodnyStoper.STAV.PoINIT:= TRUE;
				SC_P2_SpodnyStoper.ResetStep:= TRUE;
				SC_P2_SpodnyStoper.Step:= 100;
			END_IF

			//********************************************************Automatický režim****************************************************************************//
		100:
			SC_P2_SpodnyStoper.StepName:='100 - Automaticky Rezim - cakam na príchod paletky na stoper';
			SC_P2_SpodnyStoper.IdleTime.PT:= T#200ms;
			SC_P2_SpodnyStoper.AlarmTime.PT:= T#5s;

			SC_P2_SpodnyStoper.IdleTime.IN:= P2_SpodnyStoper.IN.PritomnostPaletky;

			IF P2_SpodnyStoper.KoniecCyklu THEN
				SC_P2_SpodnyStoper.ResetStep:= TRUE;
				SC_P2_SpodnyStoper.Step:= 0;
			ELSIF SC_P2_SpodnyStoper.IdleTime.Q THEN
				SC_P2_SpodnyStoper.ResetStep:= TRUE;
				SC_P2_SpodnyStoper.Step:= 101;
			END_IF

		101:
			SC_P2_SpodnyStoper.StepName:='101 - Automaticky Rezim - cakam na vyvezenie paletky na spodny stoper bunky 1';
			SC_P2_SpodnyStoper.IdleTime.PT:= T#2s;
			SC_P2_SpodnyStoper.AlarmTime.PT:= T#5s;

			SC_P2_SpodnyStoper.IdleTime.IN:= NOT P1_SpodnyStoper.IN.ZaplnenieDopravnika;

			IF P2_SpodnyStoper.KoniecCyklu THEN
				SC_P2_SpodnyStoper.ResetStep:= TRUE;
				SC_P2_SpodnyStoper.Step:= 0;
			ELSIF SC_P2_SpodnyStoper.IdleTime.Q AND P1_Dopravniky.STAV.PoINIT THEN
				SC_P2_SpodnyStoper.ResetStep:= TRUE;
				SC_P2_SpodnyStoper.Step:= 105;
			ELSIF NOT P2_SpodnyStoper.IN.PritomnostPaletky THEN
				SC_P2_SpodnyStoper.ResetStep:= TRUE;
				SC_P2_SpodnyStoper.Step:= 100;
			END_IF

		105:
			SC_P2_SpodnyStoper.StepName:='105 - Automaticky Rezim - vyvazam paletku na spodny stoper bunky 1';
			SC_P2_SpodnyStoper.IdleTime.PT:= T#200ms;
			SC_P2_SpodnyStoper.AlarmTime.PT:= T#10s;

			IF NOT SC_P2_SpodnyStoper.Switch1 THEN
				P2_SpodnyStoper.OUT.ZasunStoper:= TRUE;
				P2_SpodnyStoper.STAV.PrebiehaVyvezeniePaletky:= TRUE;
				SC_P2_SpodnyStoper.Switch1:= TRUE;
			END_IF

			IF NOT P2_SpodnyStoper.IN.PritomnostPaletky THEN
				P2_SpodnyStoper.OUT.ZasunStoper:= FALSE;
				P2_SpodnyStoper.STAV.PrebiehaVyvezeniePaletky:= FALSE;
				SC_P2_SpodnyStoper.ResetStep:= TRUE;
				SC_P2_SpodnyStoper.Step:= 100;
			END_IF

			//*******************************************************Manuálny režim*******************************************************************************//
		700:
			SC_P2_SpodnyStoper.StepName:='700 - Manualny Rezim';
			SC_P2_SpodnyStoper.IdleTime.PT:= T#8s;
			SC_P2_SpodnyStoper.AlarmTime.PT:= T#5s;

	END_CASE

END_PROGRAM

PROGRAM _EXIT
	(* Insert code here *)

END_PROGRAM
```

### Program Logical/Program/Pracovisko_2/P2_StoperZaklTesnenia (IEC)
